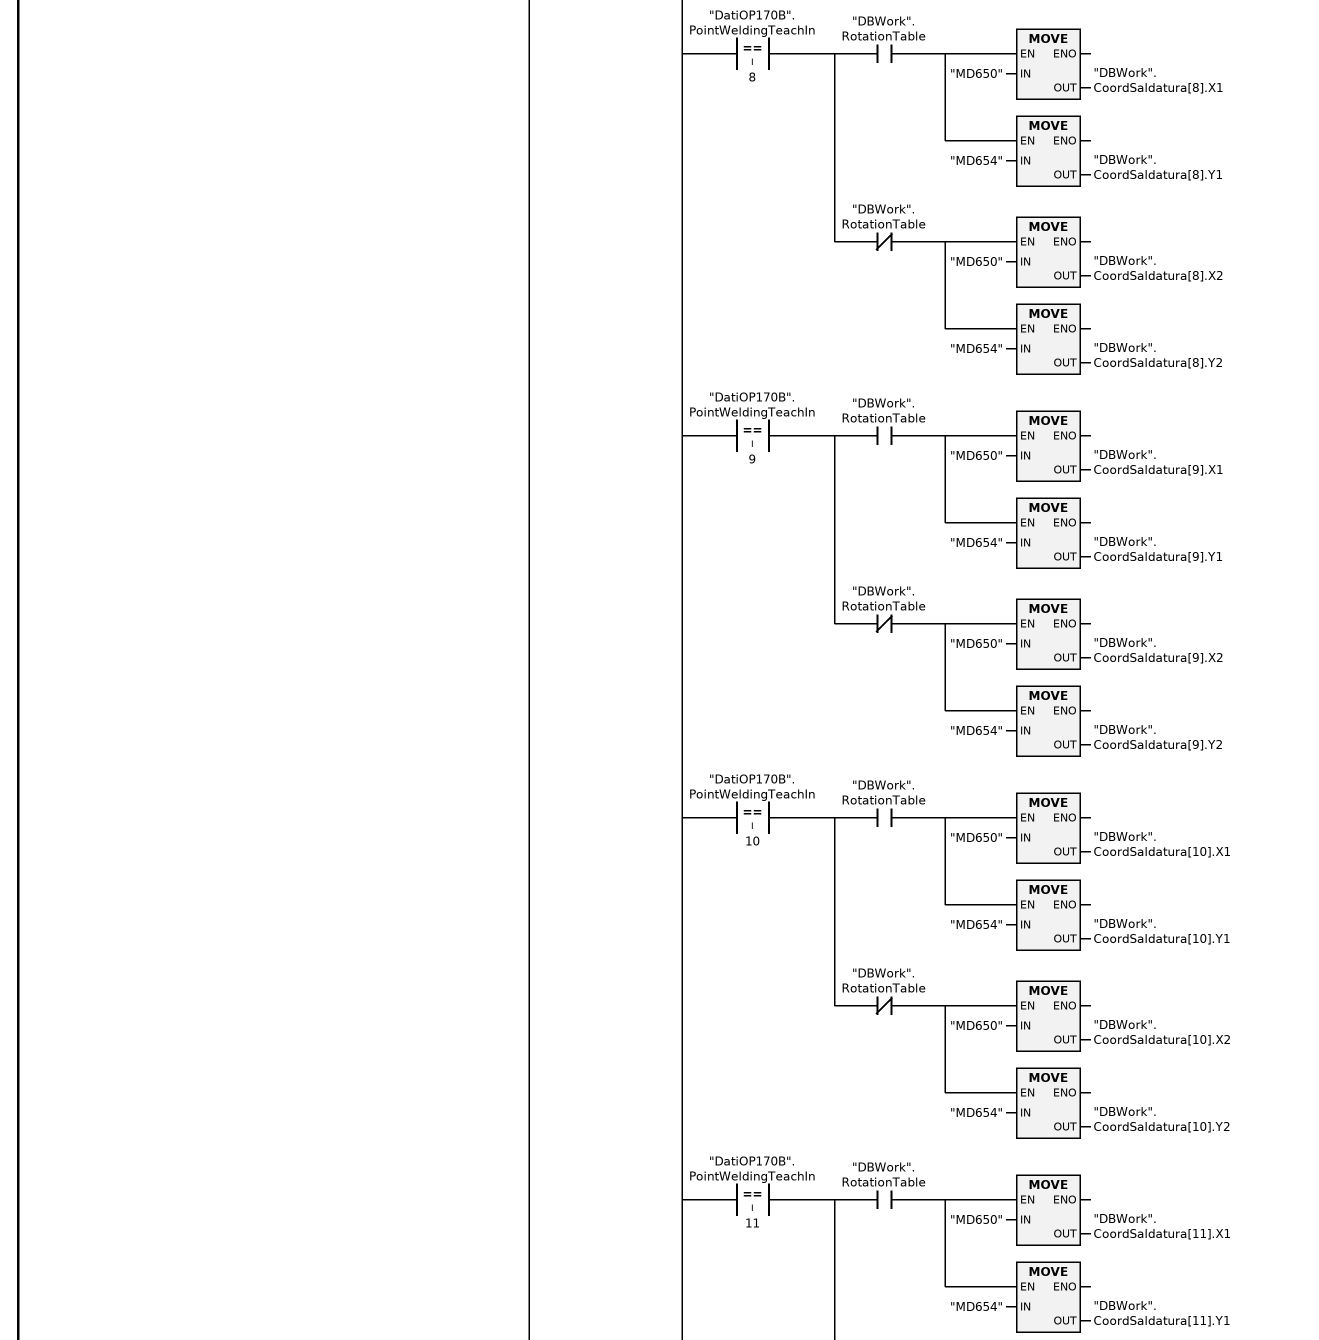
[picture p145: FC50 - TEACH-IN networks 7-7]
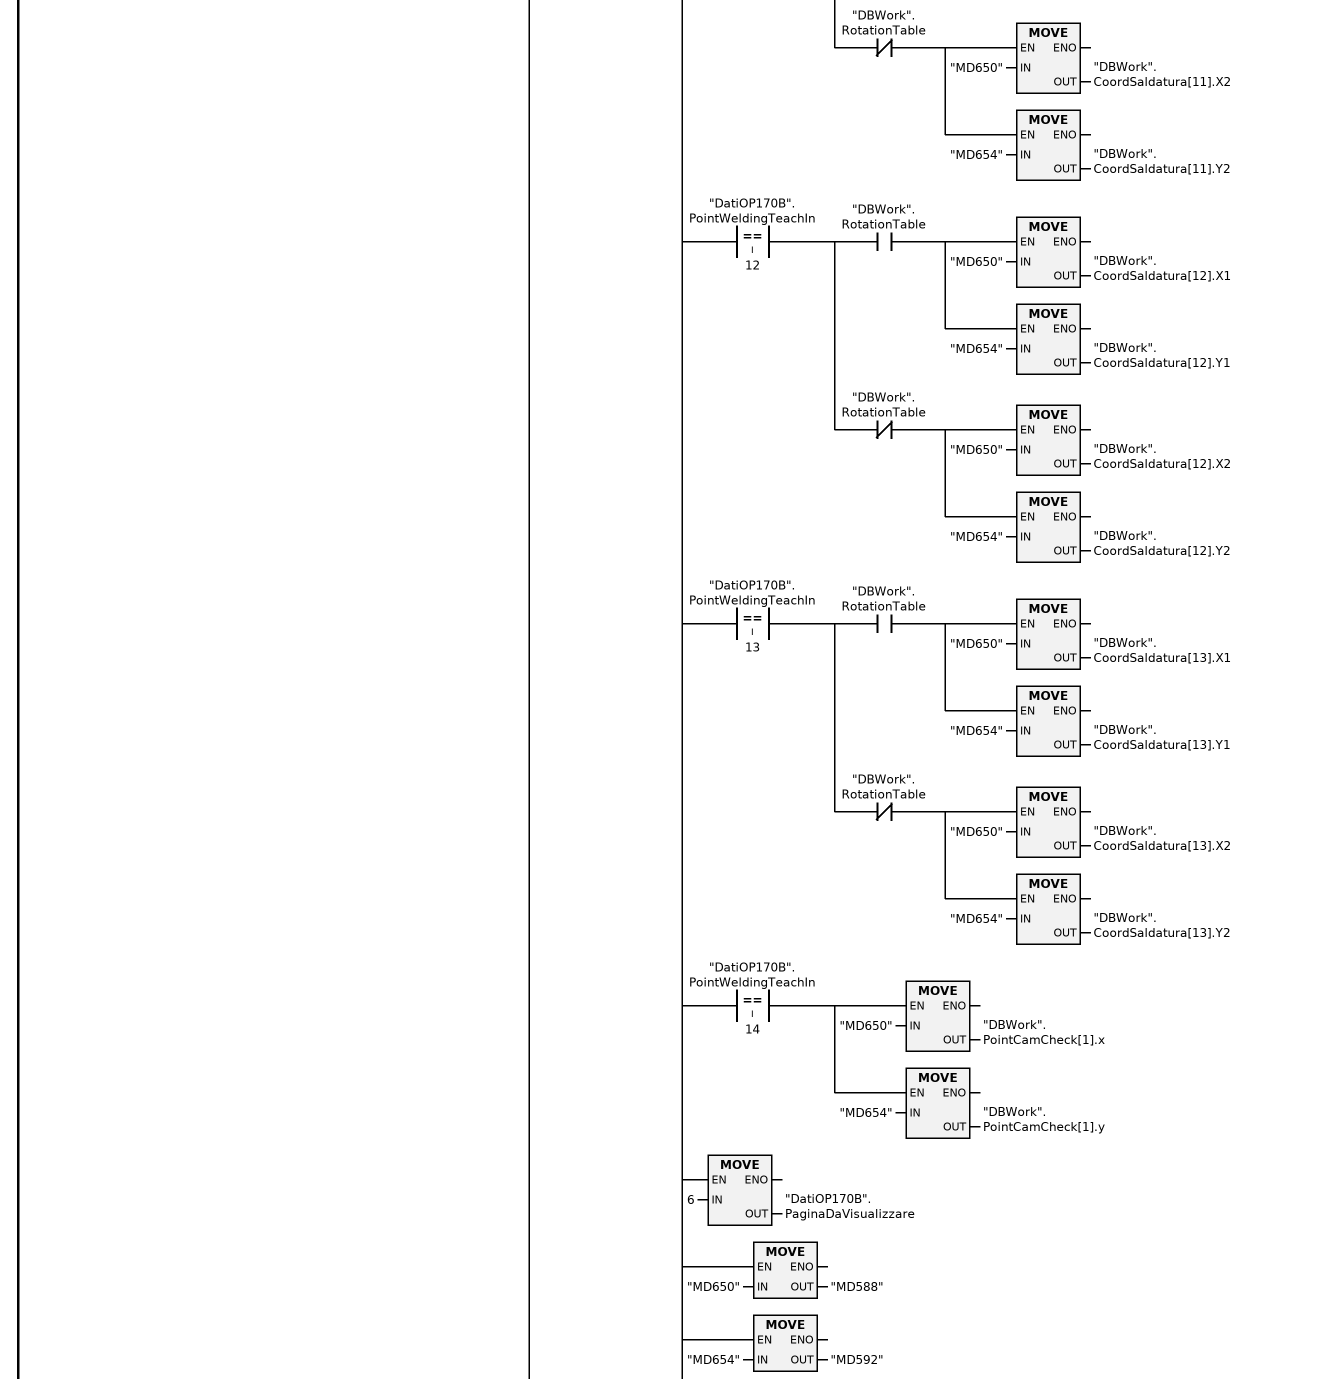
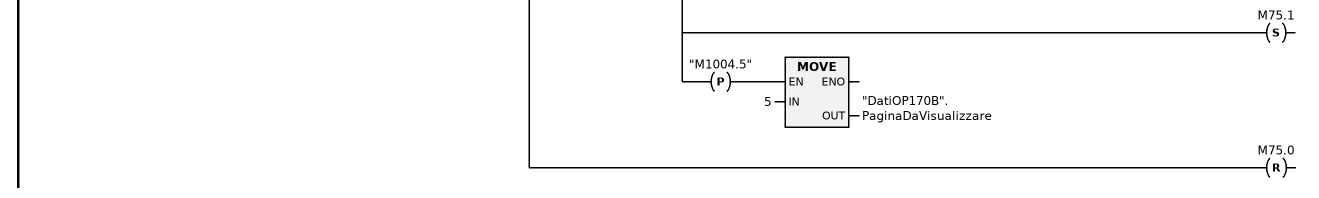
NETWORK
TITLE = Enable movement for axis on Teach-in
//move on welding point or wiev point and stored date when press teach in
//
      A     "M11.2";
      A(;
      O(;
      L     "DatiOP170B".NumeroPagina.NumeroPaginaCorrente;
      L     6;
      ==I;
      );
      O     "T63";
      );
      AN    "M346.1";
      AN    "M340.1";
      A     "M347.3";
      A     "M341.3";
      =     L 0.0;
      A     L 0.0;
      A     "T63";
      FP    "M1004.4";
      =     L 0.1;
      A     L 0.1;
      A(;
      L     "DatiOP170B".PointWeldingTeachIn;
      L     1;
      ==I;
      );
      =     L 0.2;
      A     L 0.2;
      A     "DBWork".RotationTable;
      =     L 0.3;
      A     L 0.3;
      JNB   _008;
      L     "MD650";
      T     "DBWork".CoordSaldatura[1].X1;
_008: NOP   0;
      A     L 0.3;
      JNB   _009;
      L     "MD654";
      T     "DBWork".CoordSaldatura[1].Y1;
_009: NOP   0;
      A     L 0.2;
      AN    "DBWork".RotationTable;
      =     L 0.3;
      A     L 0.3;
      JNB   _00a;
      L     "MD650";
      T     "DBWork".CoordSaldatura[1].X2;
_00a: NOP   0;
      A     L 0.3;
      JNB   _00b;
      L     "MD654";
      T     "DBWork".CoordSaldatura[1].Y2;
_00b: NOP   0;
      A     L 0.1;
      A(;
      L     "DatiOP170B".PointWeldingTeachIn;
      L     2;
      ==I;
      );
      =     L 0.2;
      A     L 0.2;
      A     "DBWork".RotationTable;
      =     L 0.3;
      A     L 0.3;
      JNB   _00c;
      L     "MD650";
      T     "DBWork".CoordSaldatura[2].X1;
_00c: NOP   0;
      A     L 0.3;
      JNB   _00d;
      L     "MD654";
      T     "DBWork".CoordSaldatura[2].Y1;
_00d: NOP   0;
      A     L 0.2;
      AN    "DBWork".RotationTable;
      =     L 0.3;
      A     L 0.3;
      JNB   _00e;
      L     "MD650";
      T     "DBWork".CoordSaldatura[2].X2;
_00e: NOP   0;
      A     L 0.3;
      JNB   _00f;
      L     "MD654";
      T     "DBWork".CoordSaldatura[2].Y2;
_00f: NOP   0;
      A     L 0.1;
      A(;
      L     "DatiOP170B".PointWeldingTeachIn;
      L     3;
      ==I;
      );
      =     L 0.2;
      A     L 0.2;
      A     "DBWork".RotationTable;
      =     L 0.3;
      A     L 0.3;
      JNB   _010;
      L     "MD650";
      T     "DBWork".CoordSaldatura[3].X1;
_010: NOP   0;
      A     L 0.3;
      JNB   _011;
      L     "MD654";
      T     "DBWork".CoordSaldatura[3].Y1;
_011: NOP   0;
      A     L 0.2;
      AN    "DBWork".RotationTable;
      =     L 0.3;
      A     L 0.3;
      JNB   _012;
      L     "MD650";
      T     "DBWork".CoordSaldatura[3].X2;
_012: NOP   0;
      A     L 0.3;
      JNB   _013;
      L     "MD654";
      T     "DBWork".CoordSaldatura[3].Y2;
_013: NOP   0;
      A     L 0.1;
      A(;
      L     "DatiOP170B".PointWeldingTeachIn;
      L     4;
      ==I;
      );
      =     L 0.2;
      A     L 0.2;
      A     "DBWork".RotationTable;
      =     L 0.3;
      A     L 0.3;
      JNB   _014;
      L     "MD650";
      T     "DBWork".CoordSaldatura[4].X1;
_014: NOP   0;
      A     L 0.3;
      JNB   _015;
      L     "MD654";
      T     "DBWork".CoordSaldatura[4].Y1;
_015: NOP   0;
      A     L 0.2;
      AN    "DBWork".RotationTable;
      =     L 0.3;
      A     L 0.3;
      JNB   _016;
      L     "MD650";
      T     "DBWork".CoordSaldatura[4].X2;
_016: NOP   0;
      A     L 0.3;
      JNB   _017;
      L     "MD654";
      T     "DBWork".CoordSaldatura[4].Y2;
_017: NOP   0;
      A     L 0.1;
      A(;
      L     "DatiOP170B".PointWeldingTeachIn;
      L     5;
      ==I;
      );
      =     L 0.2;
      A     L 0.2;
      A     "DBWork".RotationTable;
      =     L 0.3;
      A     L 0.3;
      JNB   _018;
      L     "MD650";
      T     "DBWork".CoordSaldatura[5].X1;
_018: NOP   0;
      A     L 0.3;
      JNB   _019;
      L     "MD654";
      T     "DBWork".CoordSaldatura[5].Y1;
_019: NOP   0;
      A     L 0.2;
      AN    "DBWork".RotationTable;
      =     L 0.3;
      A     L 0.3;
      JNB   _01a;
      L     "MD650";
      T     "DBWork".CoordSaldatura[5].X2;
_01a: NOP   0;
      A     L 0.3;
      JNB   _01b;
      L     "MD654";
      T     "DBWork".CoordSaldatura[5].Y2;
_01b: NOP   0;
      A     L 0.1;
      A(;
      L     "DatiOP170B".PointWeldingTeachIn;
      L     6;
      ==I;
      );
      =     L 0.2;
      A     L 0.2;
      A     "DBWork".RotationTable;
      =     L 0.3;
      A     L 0.3;
      JNB   _01c;
      L     "MD650";
      T     "DBWork".CoordSaldatura[6].X1;
_01c: NOP   0;
      A     L 0.3;
      JNB   _01d;
      L     "MD654";
      T     "DBWork".CoordSaldatura[6].Y1;
_01d: NOP   0;
      A     L 0.2;
      AN    "DBWork".RotationTable;
      =     L 0.3;
      A     L 0.3;
      JNB   _01e;
      L     "MD650";
      T     "DBWork".CoordSaldatura[6].X2;
_01e: NOP   0;
      A     L 0.3;
      JNB   _01f;
      L     "MD654";
      T     "DBWork".CoordSaldatura[6].Y2;
_01f: NOP   0;
      A     L 0.1;
      A(;
      L     "DatiOP170B".PointWeldingTeachIn;
      L     7;
      ==I;
      );
      =     L 0.2;
      A     L 0.2;
      A     "DBWork".RotationTable;
      =     L 0.3;
      A     L 0.3;
      JNB   _020;
      L     "MD650";
      T     "DBWork".CoordSaldatura[7].X1;
_020: NOP   0;
      A     L 0.3;
      JNB   _021;
      L     "MD654";
      T     "DBWork".CoordSaldatura[7].Y1;
_021: NOP   0;
      A     L 0.2;
      AN    "DBWork".RotationTable;
      =     L 0.3;
      A     L 0.3;
      JNB   _022;
      L     "MD650";
      T     "DBWork".CoordSaldatura[7].X2;
_022: NOP   0;
      A     L 0.3;
      JNB   _023;
      L     "MD654";
      T     "DBWork".CoordSaldatura[7].Y2;
_023: NOP   0;
      A     L 0.1;
      A(;
      L     "DatiOP170B".PointWeldingTeachIn;
      L     8;
      ==I;
      );
      =     L 0.2;
      A     L 0.2;
      A     "DBWork".RotationTable;
      =     L 0.3;
      A     L 0.3;
      JNB   _024;
      L     "MD650";
      T     "DBWork".CoordSaldatura[8].X1;
_024: NOP   0;
      A     L 0.3;
      JNB   _025;
      L     "MD654";
      T     "DBWork".CoordSaldatura[8].Y1;
_025: NOP   0;
      A     L 0.2;
      AN    "DBWork".RotationTable;
      =     L 0.3;
      A     L 0.3;
      JNB   _026;
      L     "MD650";
      T     "DBWork".CoordSaldatura[8].X2;
_026: NOP   0;
      A     L 0.3;
      JNB   _027;
      L     "MD654";
      T     "DBWork".CoordSaldatura[8].Y2;
_027: NOP   0;
      A     L 0.1;
      A(;
      L     "DatiOP170B".PointWeldingTeachIn;
      L     9;
      ==I;
      );
      =     L 0.2;
      A     L 0.2;
      A     "DBWork".RotationTable;
      =     L 0.3;
      A     L 0.3;
      JNB   _028;
      L     "MD650";
      T     "DBWork".CoordSaldatura[9].X1;
_028: NOP   0;
      A     L 0.3;
      JNB   _029;
      L     "MD654";
      T     "DBWork".CoordSaldatura[9].Y1;
_029: NOP   0;
      A     L 0.2;
      AN    "DBWork".RotationTable;
      =     L 0.3;
      A     L 0.3;
      JNB   _02a;
      L     "MD650";
      T     "DBWork".CoordSaldatura[9].X2;
_02a: NOP   0;
      A     L 0.3;
      JNB   _02b;
      L     "MD654";
      T     "DBWork".CoordSaldatura[9].Y2;
_02b: NOP   0;
      A     L 0.1;
      A(;
      L     "DatiOP170B".PointWeldingTeachIn;
      L     10;
      ==I;
      );
      =     L 0.2;
      A     L 0.2;
      A     "DBWork".RotationTable;
      =     L 0.3;
      A     L 0.3;
      JNB   _02c;
      L     "MD650";
      T     "DBWork".CoordSaldatura[10].X1;
_02c: NOP   0;
      A     L 0.3;
      JNB   _02d;
      L     "MD654";
      T     "DBWork".CoordSaldatura[10].Y1;
_02d: NOP   0;
      A     L 0.2;
      AN    "DBWork".RotationTable;
      =     L 0.3;
      A     L 0.3;
      JNB   _02e;
      L     "MD650";
      T     "DBWork".CoordSaldatura[10].X2;
_02e: NOP   0;
      A     L 0.3;
      JNB   _02f;
      L     "MD654";
      T     "DBWork".CoordSaldatura[10].Y2;
_02f: NOP   0;
      A     L 0.1;
      A(;
      L     "DatiOP170B".PointWeldingTeachIn;
      L     11;
      ==I;
      );
      =     L 0.2;
      A     L 0.2;
      A     "DBWork".RotationTable;
      =     L 0.3;
      A     L 0.3;
      JNB   _030;
      L     "MD650";
      T     "DBWork".CoordSaldatura[11].X1;
_030: NOP   0;
      A     L 0.3;
      JNB   _031;
      L     "MD654";
      T     "DBWork".CoordSaldatura[11].Y1;
_031: NOP   0;
      A     L 0.2;
      AN    "DBWork".RotationTable;
      =     L 0.3;
      A     L 0.3;
      JNB   _032;
      L     "MD650";
      T     "DBWork".CoordSaldatura[11].X2;
_032: NOP   0;
      A     L 0.3;
      JNB   _033;
      L     "MD654";
      T     "DBWork".CoordSaldatura[11].Y2;
_033: NOP   0;
      A     L 0.1;
      A(;
      L     "DatiOP170B".PointWeldingTeachIn;
      L     12;
      ==I;
      );
      =     L 0.2;
      A     L 0.2;
      A     "DBWork".RotationTable;
      =     L 0.3;
      A     L 0.3;
      JNB   _034;
      L     "MD650";
      T     "DBWork".CoordSaldatura[12].X1;
_034: NOP   0;
      A     L 0.3;
      JNB   _035;
      L     "MD654";
      T     "DBWork".CoordSaldatura[12].Y1;
_035: NOP   0;
      A     L 0.2;
      AN    "DBWork".RotationTable;
      =     L 0.3;
      A     L 0.3;
      JNB   _036;
      L     "MD650";
      T     "DBWork".CoordSaldatura[12].X2;
_036: NOP   0;
      A     L 0.3;
      JNB   _037;
      L     "MD654";
      T     "DBWork".CoordSaldatura[12].Y2;
_037: NOP   0;
      A     L 0.1;
      A(;
      L     "DatiOP170B".PointWeldingTeachIn;
      L     13;
      ==I;
      );
      =     L 0.2;
      A     L 0.2;
      A     "DBWork".RotationTable;
      =     L 0.3;
      A     L 0.3;
      JNB   _038;
      L     "MD650";
      T     "DBWork".CoordSaldatura[13].X1;
_038: NOP   0;
      A     L 0.3;
      JNB   _039;
      L     "MD654";
      T     "DBWork".CoordSaldatura[13].Y1;
_039: NOP   0;
      A     L 0.2;
      AN    "DBWork".RotationTable;
      =     L 0.3;
      A     L 0.3;
      JNB   _03a;
      L     "MD650";
      T     "DBWork".CoordSaldatura[13].X2;
_03a: NOP   0;
      A     L 0.3;
      JNB   _03b;
      L     "MD654";
      T     "DBWork".CoordSaldatura[13].Y2;
_03b: NOP   0;
      A     L 0.1;
      A(;
      L     "DatiOP170B".PointWeldingTeachIn;
      L     14;
      ==I;
      );
      =     L 0.2;
      A     L 0.2;
      JNB   _03c;
      L     "MD650";
      T     "DBWork".PointCamCheck[1].x;
_03c: NOP   0;
      A     L 0.2;
      JNB   _03d;
      L     "MD654";
      T     "DBWork".PointCamCheck[1].y;
_03d: NOP   0;
      A     L 0.1;
      JNB   _03e;
      L     6;
      T     "DatiOP170B".PaginaDaVisualizzare;
_03e: NOP   0;
      A     L 0.1;
      JNB   _03f;
      L     "MD650";
      T     "MD588";
_03f: NOP   0;
      A     L 0.1;
      JNB   _040;
      L     "MD654";
      T     "MD592";
_040: NOP   0;
      A     L 0.1;
      BLD   102;
      S     "M75.1";
      A     L 0.1;
      FP    "M1004.5";
      JNB   _041;
      L     5;
      T     "DatiOP170B".PaginaDaVisualizzare;
_041: NOP   0;
      A     L 0.0;
      BLD   102;
      R     "M75.0";
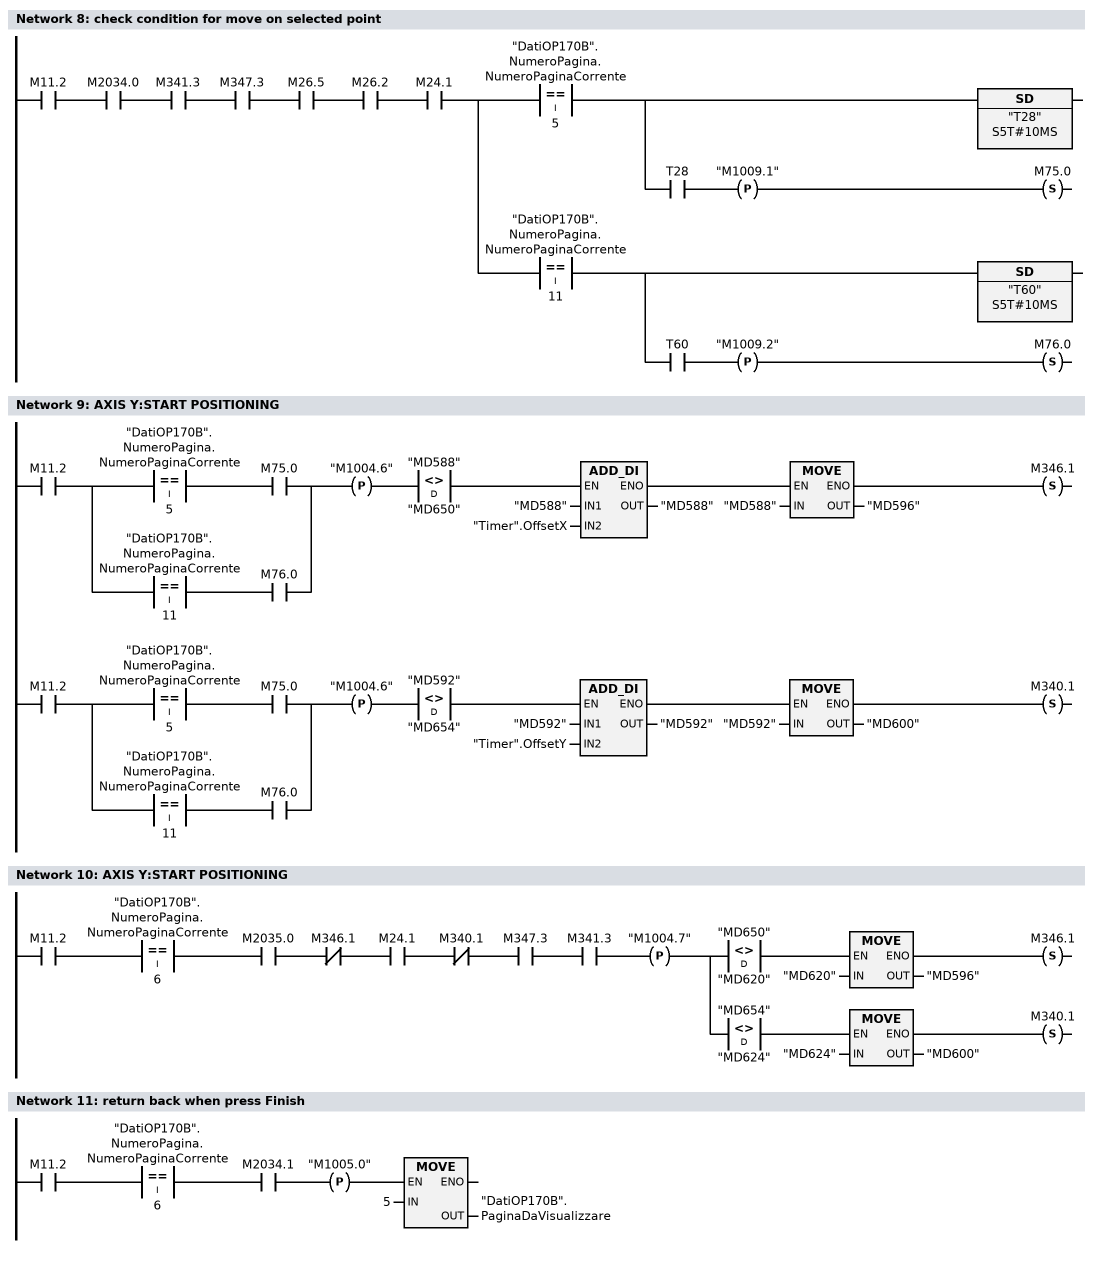
NETWORK
TITLE = check condition for move on selected point
//condition for move on selected point
      A     "M11.2";
      A     "M2034.0";
      A     "M341.3";
      A     "M347.3";
      A     "M26.5";
      A     "M26.2";
      A     "M24.1";
      =     L 1.0;
      A     L 1.0;
      A(;
      L     "DatiOP170B".NumeroPagina.NumeroPaginaCorrente;
      L     5;
      ==I;
      );
      =     L 1.1;
      A     L 1.1;
      BLD   102;
      L     S5T#10MS;
      SD    "T28";
      A     L 1.1;
      A     "T28";
      FP    "M1009.1";
      S     "M75.0";
      A     L 1.0;
      A(;
      L     "DatiOP170B".NumeroPagina.NumeroPaginaCorrente;
      L     11;
      ==I;
      );
      =     L 1.1;
      A     L 1.1;
      BLD   102;
      L     S5T#10MS;
      SD    "T60";
      A     L 1.1;
      A     "T60";
      FP    "M1009.2";
      S     "M76.0";
NETWORK
TITLE = AXIS Y:START POSITIONING
//move axis on selected point
      A     "M11.2";
      A(;
      A(;
      L     "DatiOP170B".NumeroPagina.NumeroPaginaCorrente;
      L     5;
      ==I;
      );
      A     "M75.0";
      O;
      A(;
      L     "DatiOP170B".NumeroPagina.NumeroPaginaCorrente;
      L     11;
      ==I;
      );
      A     "M76.0";
      );
      FP    "M1004.6";
      =     L 1.0;
      A(;
      A     L 1.0;
      A(;
      L     "MD588";
      L     "MD650";
      <>D;
      );
      JNB   _042;
      L     "MD588";
      L     "Timer".OffsetX;
      +D;
      T     "MD588";
      AN    OV;
      SAVE;
      CLR;
_042: A     BR;
      );
      JNB   _043;
      L     "MD588";
      T     "MD596";
      SET;
      SAVE;
      CLR;
_043: A     BR;
      S     "M346.1";
      A(;
      A     L 1.0;
      A(;
      L     "MD592";
      L     "MD654";
      <>D;
      );
      JNB   _044;
      L     "MD592";
      L     "Timer".OffsetY;
      +D;
      T     "MD592";
      AN    OV;
      SAVE;
      CLR;
_044: A     BR;
      );
      JNB   _045;
      L     "MD592";
      T     "MD600";
      SET;
      SAVE;
      CLR;
_045: A     BR;
      S     "M340.1";
NETWORK
TITLE = AXIS Y:START POSITIONING
      A     "M11.2";
      A(;
      L     "DatiOP170B".NumeroPagina.NumeroPaginaCorrente;
      L     6;
      ==I;
      );
      A     "M2035.0";
      AN    "M346.1";
      A     "M24.1";
      AN    "M340.1";
      A     "M347.3";
      A     "M341.3";
      FP    "M1004.7";
      =     L 0.0;
      A     L 0.0;
      A(;
      L     "MD650";
      L     "MD620";
      <>D;
      );
      JNB   _046;
      L     "MD620";
      T     "MD596";
      SET;
      SAVE;
      CLR;
_046: A     BR;
      S     "M346.1";
      A     L 0.0;
      A(;
      L     "MD654";
      L     "MD624";
      <>D;
      );
      JNB   _047;
      L     "MD624";
      T     "MD600";
      SET;
      SAVE;
      CLR;
_047: A     BR;
      S     "M340.1";
NETWORK
TITLE = return back when press Finish
//retirn on previus page with finish
      A     "M11.2";
      A(;
      L     "DatiOP170B".NumeroPagina.NumeroPaginaCorrente;
      L     6;
      ==I;
      );
      A     "M2034.1";
      FP    "M1005.0";
      JNB   _048;
      L     5;
      T     "DatiOP170B".PaginaDaVisualizzare;
_048: NOP   0;
END_FUNCTION

FUNCTION "FC51 - TYPE TOOL" : VOID	// FC 51
VERSION : 0.1
BEGIN
NETWORK
TITLE = 1=start read job
      A     "ChangeFunc";
      AN    "Timer".Check1;
      =     L 1.0;
      A     L 1.0;
      BLD   102;
      S     DB5.DBX 14.0;
      A     L 1.0;
      A     "Off";
      S     DB5.DBX 20.0;
NETWORK
TITLE =
NETWORK
TITLE = check if PP1 is present
//Controllo se è presente il PP1
      A(;
      AN    DB5.DBX 14.0;
      A     DB5.DBX 14.1;
      A(;
      L     DB5.DBB 16;
      L     1;
      >=I;
      );
      A(;
      L     DB5.DBB 16;
      L     5;
      <=I;
      );
      O     "Timer".Check1;
      );
      A(;
      L     "Timer".NumberVane;
      L     1;
      >=I;
      );
      A(;
      L     "Timer".NumberVane;
      L     5;
      <=I;
      );
      A(;
      A     "M15.6";
      A     "M15.7";
      O     "Timer".CheckComponent;
      );
      =     L 0.0;
      A     L 0.0;
      BLD   102;
      =     "Type_PP1";
      A     L 0.0;
      JNB   _001;
      L     10;
      T     "DBWork".NumeroSaldature;
_001: NOP   0;
NETWORK
TITLE = check if PP2 is present
//Controllo se è presente il PP2
      A(;
      AN    DB5.DBX 14.0;
      A     DB5.DBX 14.1;
      A(;
      L     DB5.DBB 16;
      L     6;
      >=I;
      );
      A(;
      L     DB5.DBB 16;
      L     10;
      <=I;
      );
      O     "Timer".Check1;
      );
      A(;
      L     "Timer".NumberVane;
      L     6;
      >=I;
      );
      A(;
      L     "Timer".NumberVane;
      L     10;
      <=I;
      );
      A(;
      A     "M15.6";
      AN    "M15.7";
      O     "Timer".CheckComponent;
      O     "On";
      );
      =     L 0.0;
      A     L 0.0;
      BLD   102;
      =     "Type_PP2";
      A     L 0.0;
      JNB   _002;
      L     11;
      T     "DBWork".NumeroSaldature;
_002: NOP   0;
NETWORK
TITLE = check if PP3 is present
//Controllo se è presente il PP3
      A(;
      AN    DB5.DBX 14.0;
      A     DB5.DBX 14.1;
      A(;
      L     DB5.DBB 16;
      L     11;
      >=I;
      );
      A(;
      L     DB5.DBB 16;
      L     15;
      <=I;
      );
      O     "Timer".Check1;
      );
      A(;
      L     "Timer".NumberVane;
      L     11;
      >=I;
      );
      A(;
      L     "Timer".NumberVane;
      L     15;
      <=I;
      );
      A(;
      AN    "M15.6";
      A     "M15.7";
      O     "Timer".CheckComponent;
      );
      =     L 0.0;
      A     L 0.0;
      BLD   102;
      =     "Type_PP3";
      A     L 0.0;
      JNB   _003;
      L     9;
      T     "DBWork".NumeroSaldature;
_003: NOP   0;
NETWORK
TITLE = check if PP4 is present
//Controllo se è presente il PP4
      A(;
      AN    DB5.DBX 14.0;
      A     DB5.DBX 14.1;
      A(;
      L     DB5.DBB 16;
      L     16;
      >=I;
      );
      A(;
      L     DB5.DBB 16;
      L     20;
      <=I;
      );
      O     "Timer".Check1;
      );
      A(;
      L     "Timer".NumberVane;
      L     16;
      >=I;
      );
      A(;
      L     "Timer".NumberVane;
      L     20;
      <=I;
      );
      A(;
      AN    "M15.6";
      AN    "M15.7";
      O     "Timer".CheckComponent;
      );
      =     L 0.0;
      A     L 0.0;
      BLD   102;
      =     "Type_PP4";
      A     L 0.0;
      JNB   _004;
      L     13;
      T     "DBWork".NumeroSaldature;
_004: NOP   0;
NETWORK
TITLE = timer for change value
      A     "ChangeFunc";
      L     S5T#1S;
      SE    "T45";
NETWORK
TITLE = load on DBWork value for weldind point PP1
//Carico sul DB Work le cordinate dei punti da saldare per il PP1
      A     "Type_PP1";
      A     "T45";
      =     L 1.0;
      A     L 1.0;
      A     "On";
      A(;
      L     "Timer".NumberVane;
      L     1;
      ==I;
      );
      =     L 1.1;
      A     L 1.1;
      JNB   _005;
      CALL  "BLKMOV" (
           SRCBLK                   := "coordinate".CoordSaldaturaPP1,
           RET_VAL                  := MW 2044,
           DSTBLK                   := "DBWork".CoordSaldatura);
_005: NOP   0;
      A     L 1.1;
      JNB   _006;
      L     "coordinate".NumeroSaldaturePP1;
      T     "DBWork".NumeroSaldature;
_006: NOP   0;
      A     L 1.1;
      JNB   _007;
      L     "coordinate".CoordinateCam_PP1[1].X;
      T     "DBWork".PointCamCheck[1].x;
_007: NOP   0;
      A     L 1.1;
      JNB   _008;
      L     "coordinate".CoordinateCam_PP1[1].Y;
      T     "DBWork".PointCamCheck[1].y;
_008: NOP   0;
      A     L 1.1;
      JNB   _009;
      L     "coordinate".CoordinateCam_PP1[2].X;
      T     "DBWork".PointCamCheck[2].x;
_009: NOP   0;
      A     L 1.1;
      JNB   _00a;
      L     "coordinate".CoordinateCam_PP1[2].Y;
      T     "DBWork".PointCamCheck[2].y;
_00a: NOP   0;
      A     L 1.1;
      JNB   _00b;
      L     "coordinate".TimeWeldingPP1[1];
      T     "DBWork".TempoSaldatura[1];
_00b: NOP   0;
      A     L 1.1;
      JNB   _00c;
      L     "coordinate".TimeWeldingPP1[2];
      T     "DBWork".TempoSaldatura[2];
_00c: NOP   0;
      A     L 1.0;
      A     "On";
      A(;
      L     "Timer".NumberVane;
      L     2;
      ==I;
      );
      =     L 1.1;
      A     L 1.1;
      JNB   _00d;
      CALL  "BLKMOV" (
           SRCBLK                   := "coordinate".CoordSaldaturaPP2,
           RET_VAL                  := MW 2044,
           DSTBLK                   := "DBWork".CoordSaldatura);
_00d: NOP   0;
      A     L 1.1;
      JNB   _00e;
      L     "coordinate".NumeroSaldaturePP2;
      T     "DBWork".NumeroSaldature;
_00e: NOP   0;
      A     L 1.1;
      JNB   _00f;
      L     "coordinate".CoordinateCam_PP2[1].X;
      T     "DBWork".PointCamCheck[1].x;
_00f: NOP   0;
      A     L 1.1;
      JNB   _010;
      L     "coordinate".CoordinateCam_PP2[1].Y;
      T     "DBWork".PointCamCheck[1].y;
_010: NOP   0;
      A     L 1.1;
      JNB   _011;
      L     "coordinate".CoordinateCam_PP2[2].X;
      T     "DBWork".PointCamCheck[2].x;
_011: NOP   0;
      A     L 1.1;
      JNB   _012;
      L     "coordinate".CoordinateCam_PP2[2].Y;
      T     "DBWork".PointCamCheck[2].y;
_012: NOP   0;
      A     L 1.1;
      JNB   _013;
      L     "coordinate".TimeWeldingPP2[1];
      T     "DBWork".TempoSaldatura[1];
_013: NOP   0;
      A     L 1.1;
      JNB   _014;
      L     "coordinate".TimeWeldingPP2[2];
      T     "DBWork".TempoSaldatura[2];
_014: NOP   0;
      A     L 1.0;
      A     "On";
      A(;
      L     "Timer".NumberVane;
      L     3;
      ==I;
      );
      =     L 1.1;
      A     L 1.1;
      JNB   _015;
      CALL  "BLKMOV" (
           SRCBLK                   := "coordinate".CoordSaldaturaPP3,
           RET_VAL                  := MW 2044,
           DSTBLK                   := "DBWork".CoordSaldatura);
_015: NOP   0;
      A     L 1.1;
      JNB   _016;
      L     "coordinate".NumeroSaldaturePP3;
      T     "DBWork".NumeroSaldature;
_016: NOP   0;
      A     L 1.1;
      JNB   _017;
      L     "coordinate".CoordinateCam_PP3[1].X;
      T     "DBWork".PointCamCheck[1].x;
_017: NOP   0;
      A     L 1.1;
      JNB   _018;
      L     "coordinate".CoordinateCam_PP3[1].Y;
      T     "DBWork".PointCamCheck[1].y;
_018: NOP   0;
      A     L 1.1;
      JNB   _019;
      L     "coordinate".CoordinateCam_PP3[2].X;
      T     "DBWork".PointCamCheck[2].x;
_019: NOP   0;
      A     L 1.1;
      JNB   _01a;
      L     "coordinate".CoordinateCam_PP3[2].Y;
      T     "DBWork".PointCamCheck[2].y;
_01a: NOP   0;
      A     L 1.1;
      JNB   _01b;
      L     "coordinate".TimeWeldingPP3[1];
      T     "DBWork".TempoSaldatura[1];
_01b: NOP   0;
      A     L 1.1;
      JNB   _01c;
      L     "coordinate".TimeWeldingPP3[2];
      T     "DBWork".TempoSaldatura[2];
_01c: NOP   0;
      A     L 1.0;
      A     "On";
      A(;
      L     "Timer".NumberVane;
      L     4;
      ==I;
      );
      =     L 1.1;
      A     L 1.1;
      JNB   _01d;
      CALL  "BLKMOV" (
           SRCBLK                   := "coordinate".CoordSaldaturaPP4,
           RET_VAL                  := MW 2044,
           DSTBLK                   := "DBWork".CoordSaldatura);
_01d: NOP   0;
      A     L 1.1;
      JNB   _01e;
      L     "coordinate".NumeroSaldaturePP4;
      T     "DBWork".NumeroSaldature;
_01e: NOP   0;
      A     L 1.1;
      JNB   _01f;
      L     "coordinate".CoordinateCam_PP4[1].X;
      T     "DBWork".PointCamCheck[1].x;
_01f: NOP   0;
      A     L 1.1;
      JNB   _020;
      L     "coordinate".CoordinateCam_PP4[1].Y;
      T     "DBWork".PointCamCheck[1].y;
_020: NOP   0;
      A     L 1.1;
      JNB   _021;
      L     "coordinate".CoordinateCam_PP4[2].X;
      T     "DBWork".PointCamCheck[2].x;
_021: NOP   0;
      A     L 1.1;
      JNB   _022;
      L     "coordinate".CoordinateCam_PP4[2].Y;
      T     "DBWork".PointCamCheck[2].y;
_022: NOP   0;
      A     L 1.1;
      JNB   _023;
      L     "coordinate".TimeWeldingPP4[1];
      T     "DBWork".TempoSaldatura[1];
_023: NOP   0;
      A     L 1.1;
      JNB   _024;
      L     "coordinate".TimeWeldingPP4[2];
      T     "DBWork".TempoSaldatura[2];
_024: NOP   0;
      A     L 1.0;
      A     "On";
      A(;
      L     "Timer".NumberVane;
      L     5;
      ==I;
      );
      =     L 1.1;
      A     L 1.1;
      JNB   _025;
      CALL  "BLKMOV" (
           SRCBLK                   := "coordinate".CoordSaldaturaPP5,
           RET_VAL                  := MW 2044,
           DSTBLK                   := "DBWork".CoordSaldatura);
_025: NOP   0;
      A     L 1.1;
      JNB   _026;
      L     "coordinate".NumeroSaldaturePP5;
      T     "DBWork".NumeroSaldature;
_026: NOP   0;
      A     L 1.1;
      JNB   _027;
      L     "coordinate".CoordinateCam_PP5[1].X;
      T     "DBWork".PointCamCheck[1].x;
_027: NOP   0;
      A     L 1.1;
      JNB   _028;
      L     "coordinate".CoordinateCam_PP5[1].Y;
      T     "DBWork".PointCamCheck[1].y;
_028: NOP   0;
      A     L 1.1;
      JNB   _029;
      L     "coordinate".CoordinateCam_PP5[2].X;
      T     "DBWork".PointCamCheck[2].x;
_029: NOP   0;
      A     L 1.1;
      JNB   _02a;
      L     "coordinate".CoordinateCam_PP5[2].Y;
      T     "DBWork".PointCamCheck[2].y;
_02a: NOP   0;
      A     L 1.1;
      JNB   _02b;
      L     "coordinate".TimeWeldingPP5[1];
      T     "DBWork".TempoSaldatura[1];
_02b: NOP   0;
      A     L 1.1;
      JNB   _02c;
      L     "coordinate".TimeWeldingPP5[2];
      T     "DBWork".TempoSaldatura[2];
_02c: NOP   0;
NETWORK
TITLE = load on DBWork value for weldind point PP2
//Carico sul DB Work le cordinate dei punti da saldare per il PP2
      A     "Type_PP2";
      A     "T45";
      =     L 1.0;
      A     L 1.0;
      A     "On";
      A(;
      L     "Timer".NumberVane;
      L     6;
      ==I;
      );
      =     L 1.1;
      A     L 1.1;
      JNB   _02d;
      CALL  "BLKMOV" (
           SRCBLK                   := "coordinate".CoordSaldaturaPP6,
           RET_VAL                  := MW 2044,
           DSTBLK                   := "DBWork".CoordSaldatura);
_02d: NOP   0;
      A     L 1.1;
      JNB   _02e;
      L     "coordinate".NumeroSaldaturePP6;
      T     "DBWork".NumeroSaldature;
_02e: NOP   0;
      A     L 1.1;
      JNB   _02f;
      L     "coordinate".CoordinateCam_PP6[1].X;
      T     "DBWork".PointCamCheck[1].x;
_02f: NOP   0;
      A     L 1.1;
      JNB   _030;
      L     "coordinate".CoordinateCam_PP6[1].Y;
      T     "DBWork".PointCamCheck[1].y;
_030: NOP   0;
      A     L 1.1;
      JNB   _031;
      L     "coordinate".TimeWeldingPP6[1];
      T     "DBWork".TempoSaldatura[1];
_031: NOP   0;
      A     L 1.1;
      JNB   _032;
      L     "coordinate".TimeWeldingPP6[2];
      T     "DBWork".TempoSaldatura[2];
_032: NOP   0;
      A     L 1.0;
      A     "On";
      A(;
      L     "Timer".NumberVane;
      L     7;
      ==I;
      );
      =     L 1.1;
      A     L 1.1;
      JNB   _033;
      CALL  "BLKMOV" (
           SRCBLK                   := "coordinate".CoordSaldaturaPP7,
           RET_VAL                  := MW 2044,
           DSTBLK                   := "DBWork".CoordSaldatura);
_033: NOP   0;
      A     L 1.1;
      JNB   _034;
      L     "coordinate".NumeroSaldaturePP7;
      T     "DBWork".NumeroSaldature;
_034: NOP   0;
      A     L 1.1;
      JNB   _035;
      L     "coordinate".CoordinateCam_PP7[1].X;
      T     "DBWork".PointCamCheck[1].x;
_035: NOP   0;
      A     L 1.1;
      JNB   _036;
      L     "coordinate".CoordinateCam_PP7[1].Y;
      T     "DBWork".PointCamCheck[1].y;
_036: NOP   0;
      A     L 1.1;
      JNB   _037;
      L     "coordinate".TimeWeldingPP7[1];
      T     "DBWork".TempoSaldatura[1];
_037: NOP   0;
      A     L 1.1;
      JNB   _038;
      L     "coordinate".TimeWeldingPP7[2];
      T     "DBWork".TempoSaldatura[2];
_038: NOP   0;
      A     L 1.0;
      A     "On";
      A(;
      L     "Timer".NumberVane;
      L     8;
      ==I;
      );
      =     L 1.1;
      A     L 1.1;
      JNB   _039;
      CALL  "BLKMOV" (
           SRCBLK                   := "coordinate".CoordSaldaturaPP8,
           RET_VAL                  := MW 2044,
           DSTBLK                   := "DBWork".CoordSaldatura);
_039: NOP   0;
      A     L 1.1;
      JNB   _03a;
      L     "coordinate".NumeroSaldaturePP8;
      T     "DBWork".NumeroSaldature;
_03a: NOP   0;
      A     L 1.1;
      JNB   _03b;
      L     "coordinate".CoordinateCam_PP8[1].X;
      T     "DBWork".PointCamCheck[1].x;
_03b: NOP   0;
      A     L 1.1;
      JNB   _03c;
      L     "coordinate".CoordinateCam_PP8[1].Y;
      T     "DBWork".PointCamCheck[1].y;
_03c: NOP   0;
      A     L 1.1;
      JNB   _03d;
      L     "coordinate".TimeWeldingPP8[1];
      T     "DBWork".TempoSaldatura[1];
_03d: NOP   0;
      A     L 1.1;
      JNB   _03e;
      L     "coordinate".TimeWeldingPP8[2];
      T     "DBWork".TempoSaldatura[2];
_03e: NOP   0;
      A     L 1.0;
      A     "On";
      A(;
      L     "Timer".NumberVane;
      L     9;
      ==I;
      );
      =     L 1.1;
      A     L 1.1;
      JNB   _03f;
      CALL  "BLKMOV" (
           SRCBLK                   := "coordinate".CoordSaldaturaPP9,
           RET_VAL                  := MW 2044,
           DSTBLK                   := "DBWork".CoordSaldatura);
_03f: NOP   0;
      A     L 1.1;
      JNB   _040;
      L     "coordinate".NumeroSaldaturePP9;
      T     "DBWork".NumeroSaldature;
_040: NOP   0;
      A     L 1.1;
      JNB   _041;
      L     "coordinate".CoordinateCam_PP9[1].X;
      T     "DBWork".PointCamCheck[1].x;
_041: NOP   0;
      A     L 1.1;
      JNB   _042;
      L     "coordinate".CoordinateCam_PP9[1].Y;
      T     "DBWork".PointCamCheck[1].y;
_042: NOP   0;
      A     L 1.1;
      JNB   _043;
      L     "coordinate".TimeWeldingPP9[1];
      T     "DBWork".TempoSaldatura[1];
_043: NOP   0;
      A     L 1.1;
      JNB   _044;
      L     "coordinate".TimeWeldingPP9[2];
      T     "DBWork".TempoSaldatura[2];
_044: NOP   0;
      A     L 1.0;
      A     "On";
      A(;
      L     "Timer".NumberVane;
      L     10;
      ==I;
      );
      =     L 1.1;
      A     L 1.1;
      JNB   _045;
      CALL  "BLKMOV" (
           SRCBLK                   := "coordinate".CoordSaldaturaPP10,
           RET_VAL                  := MW 2044,
           DSTBLK                   := "DBWork".CoordSaldatura);
_045: NOP   0;
      A     L 1.1;
      JNB   _046;
      L     "coordinate".NumeroSaldaturePP10;
      T     "DBWork".NumeroSaldature;
_046: NOP   0;
      A     L 1.1;
      JNB   _047;
      L     "coordinate".CoordinateCam_PP10[1].X;
      T     "DBWork".PointCamCheck[1].x;
_047: NOP   0;
      A     L 1.1;
      JNB   _048;
      L     "coordinate".CoordinateCam_PP10[1].Y;
      T     "DBWork".PointCamCheck[1].y;
_048: NOP   0;
      A     L 1.1;
      JNB   _049;
      L     "coordinate".TimeWeldingPP10[1];
      T     "DBWork".TempoSaldatura[1];
_049: NOP   0;
      A     L 1.1;
      JNB   _04a;
      L     "coordinate".TimeWeldingPP10[2];
      T     "DBWork".TempoSaldatura[2];
_04a: NOP   0;
NETWORK
TITLE = load on DBWork value for weldind point PP3
//Carico sul DB Work le cordinate dei punti da saldare per il PP3
      A     "Type_PP3";
      A     "T45";
      =     L 1.0;
      A     L 1.0;
      A     "On";
      A(;
      L     "Timer".NumberVane;
      L     11;
      ==I;
      );
      =     L 1.1;
      A     L 1.1;
      JNB   _04b;
      CALL  "BLKMOV" (
           SRCBLK                   := "coordinate".CoordSaldaturaPP11,
           RET_VAL                  := MW 2044,
           DSTBLK                   := "DBWork".CoordSaldatura);
_04b: NOP   0;
      A     L 1.1;
      JNB   _04c;
      L     "coordinate".NumeroSaldaturePP11;
      T     "DBWork".NumeroSaldature;
_04c: NOP   0;
      A     L 1.1;
      JNB   _04d;
      L     "coordinate".CoordinateCam_PP11[1].X;
      T     "DBWork".PointCamCheck[1].x;
_04d: NOP   0;
      A     L 1.1;
      JNB   _04e;
      L     "coordinate".CoordinateCam_PP11[1].Y;
      T     "DBWork".PointCamCheck[1].y;
_04e: NOP   0;
      A     L 1.1;
      JNB   _04f;
      L     "coordinate".TimeWeldingPP11[1];
      T     "DBWork".TempoSaldatura[1];
_04f: NOP   0;
      A     L 1.1;
      JNB   _050;
      L     "coordinate".TimeWeldingPP11[2];
      T     "DBWork".TempoSaldatura[2];
_050: NOP   0;
      A     L 1.0;
      A     "On";
      A(;
      L     "Timer".NumberVane;
      L     12;
      ==I;
      );
      =     L 1.1;
      A     L 1.1;
      JNB   _051;
      CALL  "BLKMOV" (
           SRCBLK                   := "coordinate".CoordSaldaturaPP12,
           RET_VAL                  := MW 2044,
           DSTBLK                   := "DBWork".CoordSaldatura);
_051: NOP   0;
      A     L 1.1;
      JNB   _052;
      L     "coordinate".NumeroSaldaturePP12;
      T     "DBWork".NumeroSaldature;
_052: NOP   0;
      A     L 1.1;
      JNB   _053;
      L     "coordinate".NumeroSaldaturePP12;
      T     "DBWork".NumeroSaldature;
_053: NOP   0;
      A     L 1.1;
      JNB   _054;
      L     "coordinate".CoordinateCam_PP12[1].X;
      T     "DBWork".PointCamCheck[1].x;
_054: NOP   0;
      A     L 1.1;
      JNB   _055;
      L     "coordinate".CoordinateCam_PP12[1].Y;
      T     "DBWork".PointCamCheck[1].y;
_055: NOP   0;
      A     L 1.1;
      JNB   _056;
      L     "coordinate".TimeWeldingPP12[2];
      T     "DBWork".TempoSaldatura[2];
_056: NOP   0;
      A     L 1.0;
      A     "On";
      A(;
      L     "Timer".NumberVane;
      L     13;
      ==I;
      );
      =     L 1.1;
      A     L 1.1;
      JNB   _057;
      CALL  "BLKMOV" (
           SRCBLK                   := "coordinate".CoordSaldaturaPP13,
           RET_VAL                  := MW 2044,
           DSTBLK                   := "DBWork".CoordSaldatura);
_057: NOP   0;
      A     L 1.1;
      JNB   _058;
      L     "coordinate".NumeroSaldaturePP13;
      T     "DBWork".NumeroSaldature;
_058: NOP   0;
      A     L 1.1;
      JNB   _059;
      L     "coordinate".NumeroSaldaturePP13;
      T     "DBWork".NumeroSaldature;
_059: NOP   0;
      A     L 1.1;
      JNB   _05a;
      L     "coordinate".CoordinateCam_PP13[1].X;
      T     "DBWork".PointCamCheck[1].x;
_05a: NOP   0;
      A     L 1.1;
      JNB   _05b;
      L     "coordinate".CoordinateCam_PP13[1].Y;
      T     "DBWork".PointCamCheck[1].y;
_05b: NOP   0;
      A     L 1.1;
      JNB   _05c;
      L     "coordinate".TimeWeldingPP13[2];
      T     "DBWork".TempoSaldatura[2];
_05c: NOP   0;
      A     L 1.0;
      A     "On";
      A(;
      L     "Timer".NumberVane;
      L     14;
      ==I;
      );
      =     L 1.1;
      A     L 1.1;
      JNB   _05d;
      CALL  "BLKMOV" (
           SRCBLK                   := "coordinate".CoordSaldaturaPP14,
           RET_VAL                  := MW 2044,
           DSTBLK                   := "DBWork".CoordSaldatura);
_05d: NOP   0;
      A     L 1.1;
      JNB   _05e;
      L     "coordinate".NumeroSaldaturePP14;
      T     "DBWork".NumeroSaldature;
_05e: NOP   0;
      A     L 1.1;
      JNB   _05f;
      L     "coordinate".NumeroSaldaturePP14;
      T     "DBWork".NumeroSaldature;
_05f: NOP   0;
      A     L 1.1;
      JNB   _060;
      L     "coordinate".NumeroSaldaturePP14;
      T     "DBWork".NumeroSaldature;
_060: NOP   0;
      A     L 1.1;
      JNB   _061;
      L     "coordinate".CoordinateCam_PP14[1].X;
      T     "DBWork".PointCamCheck[1].x;
_061: NOP   0;
      A     L 1.1;
      JNB   _062;
      L     "coordinate".CoordinateCam_PP14[1].Y;
      T     "DBWork".PointCamCheck[1].y;
_062: NOP   0;
      A     L 1.1;
      JNB   _063;
      L     "coordinate".TimeWeldingPP14[2];
      T     "DBWork".TempoSaldatura[2];
_063: NOP   0;
      A     L 1.0;
      A     "On";
      A(;
      L     "Timer".NumberVane;
      L     15;
      ==I;
      );
      =     L 1.1;
      A     L 1.1;
      JNB   _064;
      CALL  "BLKMOV" (
           SRCBLK                   := "coordinate".CoordSaldaturaPP15,
           RET_VAL                  := MW 2044,
           DSTBLK                   := "DBWork".CoordSaldatura);
_064: NOP   0;
      A     L 1.1;
      JNB   _065;
      L     "coordinate".NumeroSaldaturePP15;
      T     "DBWork".NumeroSaldature;
_065: NOP   0;
      A     L 1.1;
      JNB   _066;
      L     "coordinate".NumeroSaldaturePP15;
      T     "DBWork".NumeroSaldature;
_066: NOP   0;
      A     L 1.1;
      JNB   _067;
      L     "coordinate".NumeroSaldaturePP15;
      T     "DBWork".NumeroSaldature;
_067: NOP   0;
      A     L 1.1;
      JNB   _068;
      L     "coordinate".NumeroSaldaturePP15;
      T     "DBWork".NumeroSaldature;
_068: NOP   0;
      A     L 1.1;
      JNB   _069;
      L     "coordinate".CoordinateCam_PP15[1].X;
      T     "DBWork".PointCamCheck[1].x;
_069: NOP   0;
      A     L 1.1;
      JNB   _06a;
      L     "coordinate".CoordinateCam_PP15[1].Y;
      T     "DBWork".PointCamCheck[1].y;
_06a: NOP   0;
      A     L 1.1;
      JNB   _06b;
      L     "coordinate".TimeWeldingPP15[2];
      T     "DBWork".TempoSaldatura[2];
_06b: NOP   0;
NETWORK
TITLE = load on DBWork value for weldind point PP4
//Carico sul DB Work le cordinate dei punti da saldare per il PP4
      A     "Type_PP4";
      A     "T45";
      =     L 1.0;
      A     L 1.0;
      A     "On";
      A(;
      L     "Timer".NumberVane;
      L     16;
      ==I;
      );
      =     L 1.1;
      A     L 1.1;
      JNB   _06c;
      CALL  "BLKMOV" (
           SRCBLK                   := "coordinate".CoordSaldaturaPP16,
           RET_VAL                  := MW 2044,
           DSTBLK                   := "DBWork".CoordSaldatura);
_06c: A     BR;
      S     M 465.0;
      A     L 1.1;
      JNB   _06d;
      L     "coordinate".NumeroSaldaturePP16;
      T     "DBWork".NumeroSaldature;
_06d: NOP   0;
      A     L 1.1;
      JNB   _06e;
      L     "coordinate".CoordinateCam_PP16[1].X;
      T     "DBWork".PointCamCheck[1].x;
_06e: NOP   0;
      A     L 1.1;
      JNB   _06f;
      L     "coordinate".CoordinateCam_PP16[1].Y;
      T     "DBWork".PointCamCheck[1].y;
_06f: NOP   0;
      A     L 1.1;
      JNB   _070;
      L     "coordinate".TimeWeldingPP16[1];
      T     "DBWork".TempoSaldatura[1];
_070: NOP   0;
      A     L 1.1;
      JNB   _071;
      L     "coordinate".TimeWeldingPP16[2];
      T     "DBWork".TempoSaldatura[2];
_071: NOP   0;
      A     L 1.0;
      A     "On";
      A(;
      L     "Timer".NumberVane;
      L     17;
      ==I;
      );
      =     L 1.1;
      A     L 1.1;
      JNB   _072;
      CALL  "BLKMOV" (
           SRCBLK                   := "coordinate".CoordSaldaturaPP17,
           RET_VAL                  := MW 2044,
           DSTBLK                   := "DBWork".CoordSaldatura);
_072: NOP   0;
      A     L 1.1;
      JNB   _073;
      L     "coordinate".NumeroSaldaturePP17;
      T     "DBWork".NumeroSaldature;
_073: NOP   0;
      A     L 1.1;
      JNB   _074;
      L     "coordinate".CoordinateCam_PP17[1].X;
      T     "DBWork".PointCamCheck[1].x;
_074: NOP   0;
      A     L 1.1;
      JNB   _075;
      L     "coordinate".CoordinateCam_PP17[1].Y;
      T     "DBWork".PointCamCheck[1].y;
_075: NOP   0;
      A     L 1.1;
      JNB   _076;
      L     "coordinate".TimeWeldingPP17[1];
      T     "DBWork".TempoSaldatura[1];
_076: NOP   0;
      A     L 1.1;
      JNB   _077;
      L     "coordinate".TimeWeldingPP17[2];
      T     "DBWork".TempoSaldatura[2];
_077: NOP   0;
      A     L 1.0;
      A     "On";
      A(;
      L     "Timer".NumberVane;
      L     18;
      ==I;
      );
      =     L 1.1;
      A     L 1.1;
      JNB   _078;
      CALL  "BLKMOV" (
           SRCBLK                   := "coordinate".CoordSaldaturaPP18,
           RET_VAL                  := MW 2044,
           DSTBLK                   := "DBWork".CoordSaldatura);
_078: NOP   0;
      A     L 1.1;
      JNB   _079;
      L     "coordinate".NumeroSaldaturePP18;
      T     "DBWork".NumeroSaldature;
_079: NOP   0;
      A     L 1.1;
      JNB   _07a;
      L     "coordinate".CoordinateCam_PP18[1].X;
      T     "DBWork".PointCamCheck[1].x;
_07a: NOP   0;
      A     L 1.1;
      JNB   _07b;
      L     "coordinate".CoordinateCam_PP18[1].Y;
      T     "DBWork".PointCamCheck[1].y;
_07b: NOP   0;
      A     L 1.1;
      JNB   _07c;
      L     "coordinate".TimeWeldingPP18[1];
      T     "DBWork".TempoSaldatura[1];
_07c: NOP   0;
      A     L 1.1;
      JNB   _07d;
      L     "coordinate".TimeWeldingPP18[2];
      T     "DBWork".TempoSaldatura[2];
_07d: NOP   0;
      A     L 1.0;
      A     "On";
      A(;
      L     "Timer".NumberVane;
      L     19;
      ==I;
      );
      =     L 1.1;
      A     L 1.1;
      JNB   _07e;
      CALL  "BLKMOV" (
           SRCBLK                   := "coordinate".CoordSaldaturaPP19,
           RET_VAL                  := MW 2044,
           DSTBLK                   := "DBWork".CoordSaldatura);
_07e: NOP   0;
      A     L 1.1;
      JNB   _07f;
      L     "coordinate".NumeroSaldaturePP19;
      T     "DBWork".NumeroSaldature;
_07f: NOP   0;
      A     L 1.1;
      JNB   _080;
      L     "coordinate".CoordinateCam_PP19[1].X;
      T     "DBWork".PointCamCheck[1].x;
_080: NOP   0;
      A     L 1.1;
      JNB   _081;
      L     "coordinate".CoordinateCam_PP19[1].Y;
      T     "DBWork".PointCamCheck[1].y;
_081: NOP   0;
      A     L 1.1;
      JNB   _082;
      L     "coordinate".TimeWeldingPP19[1];
      T     "DBWork".TempoSaldatura[1];
_082: NOP   0;
      A     L 1.1;
      JNB   _083;
      L     "coordinate".TimeWeldingPP19[2];
      T     "DBWork".TempoSaldatura[2];
_083: NOP   0;
      A     L 1.0;
      A     "On";
      A(;
      L     "Timer".NumberVane;
      L     20;
      ==I;
      );
      =     L 1.1;
      A     L 1.1;
      JNB   _084;
      CALL  "BLKMOV" (
           SRCBLK                   := "coordinate".CoordSaldaturaPP20,
           RET_VAL                  := MW 2044,
           DSTBLK                   := "DBWork".CoordSaldatura);
_084: NOP   0;
      A     L 1.1;
      JNB   _085;
      L     "coordinate".NumeroSaldaturePP20;
      T     "DBWork".NumeroSaldature;
_085: NOP   0;
      A     L 1.1;
      JNB   _086;
      L     "coordinate".CoordinateCam_PP20[1].X;
      T     "DBWork".PointCamCheck[1].x;
_086: NOP   0;
      A     L 1.1;
      JNB   _087;
      L     "coordinate".CoordinateCam_PP20[1].Y;
      T     "DBWork".PointCamCheck[1].y;
_087: NOP   0;
      A     L 1.1;
      JNB   _088;
      L     "coordinate".TimeWeldingPP20[1];
      T     "DBWork".TempoSaldatura[1];
_088: NOP   0;
      A     L 1.1;
      JNB   _089;
      L     "coordinate".TimeWeldingPP20[2];
      T     "DBWork".TempoSaldatura[2];
_089: NOP   0;
NETWORK
TITLE =
NETWORK
TITLE = TeachIn finish, save value for PP1
//Salvo sul Db Coordinate  i nuovi valori impostati con il teachIn per PP1.
      A     "Type_PP1";
      A     "M75.1";
      =     L 1.0;
      A     L 1.0;
      A     "On";
      A(;
      L     "Timer".NumberVane;
      L     1;
      ==I;
      );
      =     L 1.1;
      A     L 1.1;
      JNB   _08a;
      CALL  "BLKMOV" (
           SRCBLK                   := "DBWork".CoordSaldatura,
           RET_VAL                  := MW 2044,
           DSTBLK                   := "coordinate".CoordSaldaturaPP1);
_08a: A     BR;
      R     "M75.1";
      A     L 1.1;
      JNB   _08b;
      L     "DBWork".PointCamCheck[1].x;
      T     "coordinate".CoordinateCam_PP1[1].X;
_08b: NOP   0;
      A     L 1.1;
      JNB   _08c;
      L     "DBWork".PointCamCheck[1].y;
      T     "coordinate".CoordinateCam_PP1[1].Y;
_08c: NOP   0;
      A     L 1.0;
      A     "On";
      A(;
      L     "Timer".NumberVane;
      L     2;
      ==I;
      );
      =     L 1.1;
      A     L 1.1;
      JNB   _08d;
      CALL  "BLKMOV" (
           SRCBLK                   := "DBWork".CoordSaldatura,
           RET_VAL                  := MW 2044,
           DSTBLK                   := "coordinate".CoordSaldaturaPP2);
_08d: A     BR;
      R     "M75.1";
      A     L 1.1;
      JNB   _08e;
      L     "DBWork".PointCamCheck[1].x;
      T     "coordinate".CoordinateCam_PP2[1].X;
_08e: NOP   0;
      A     L 1.1;
      JNB   _08f;
      L     "DBWork".PointCamCheck[1].y;
      T     "coordinate".CoordinateCam_PP2[1].Y;
_08f: NOP   0;
      A     L 1.0;
      A     "On";
      A(;
      L     "Timer".NumberVane;
      L     3;
      ==I;
      );
      =     L 1.1;
      A     L 1.1;
      JNB   _090;
      CALL  "BLKMOV" (
           SRCBLK                   := "DBWork".CoordSaldatura,
           RET_VAL                  := MW 2044,
           DSTBLK                   := "coordinate".CoordSaldaturaPP3);
_090: A     BR;
      R     "M75.1";
      A     L 1.1;
      JNB   _091;
      L     "DBWork".PointCamCheck[1].x;
      T     "coordinate".CoordinateCam_PP3[1].X;
_091: NOP   0;
      A     L 1.1;
      JNB   _092;
      L     "DBWork".PointCamCheck[1].y;
      T     "coordinate".CoordinateCam_PP3[1].Y;
_092: NOP   0;
      A     L 1.0;
      A     "On";
      A(;
      L     "Timer".NumberVane;
      L     4;
      ==I;
      );
      =     L 1.1;
      A     L 1.1;
      JNB   _093;
      CALL  "BLKMOV" (
           SRCBLK                   := "DBWork".CoordSaldatura,
           RET_VAL                  := MW 2044,
           DSTBLK                   := "coordinate".CoordSaldaturaPP4);
_093: A     BR;
      R     "M75.1";
      A     L 1.1;
      JNB   _094;
      L     "DBWork".PointCamCheck[1].x;
      T     "coordinate".CoordinateCam_PP4[1].X;
_094: NOP   0;
      A     L 1.1;
      JNB   _095;
      L     "DBWork".PointCamCheck[1].y;
      T     "coordinate".CoordinateCam_PP4[1].Y;
_095: NOP   0;
      A     L 1.0;
      A     "On";
      A(;
      L     "Timer".NumberVane;
      L     5;
      ==I;
      );
      =     L 1.1;
      A     L 1.1;
      JNB   _096;
      CALL  "BLKMOV" (
           SRCBLK                   := "DBWork".CoordSaldatura,
           RET_VAL                  := MW 2044,
           DSTBLK                   := "coordinate".CoordSaldaturaPP5);
_096: A     BR;
      R     "M75.1";
      A     L 1.1;
      JNB   _097;
      L     "DBWork".PointCamCheck[1].x;
      T     "coordinate".CoordinateCam_PP5[1].X;
_097: NOP   0;
      A     L 1.1;
      JNB   _098;
      L     "DBWork".PointCamCheck[1].y;
      T     "coordinate".CoordinateCam_PP5[1].Y;
_098: NOP   0;
NETWORK
TITLE = TeachIn finish, save value for PP2
//Salvo sul Db Coordinate  i nuovi valori impostati con il teachIn per PP2.
      A     "Type_PP2";
      A     "M75.1";
      =     L 1.0;
      A     L 1.0;
      A     "On";
      A(;
      L     "Timer".NumberVane;
      L     6;
      ==I;
      );
      =     L 1.1;
      A     L 1.1;
      JNB   _099;
      CALL  "BLKMOV" (
           SRCBLK                   := "DBWork".CoordSaldatura,
           RET_VAL                  := MW 2044,
           DSTBLK                   := "coordinate".CoordSaldaturaPP6);
_099: A     BR;
      R     "M75.1";
      A     L 1.1;
      JNB   _09a;
      L     "DBWork".PointCamCheck[1].x;
      T     "coordinate".CoordinateCam_PP6[1].X;
_09a: NOP   0;
      A     L 1.1;
      JNB   _09b;
      L     "DBWork".PointCamCheck[1].y;
      T     "coordinate".CoordinateCam_PP6[1].Y;
_09b: NOP   0;
      A     L 1.0;
      A     "On";
      A(;
      L     "Timer".NumberVane;
      L     7;
      ==I;
      );
      =     L 1.1;
      A     L 1.1;
      JNB   _09c;
      CALL  "BLKMOV" (
           SRCBLK                   := "DBWork".CoordSaldatura,
           RET_VAL                  := MW 2044,
           DSTBLK                   := "coordinate".CoordSaldaturaPP7);
_09c: A     BR;
      R     "M75.1";
      A     L 1.1;
      JNB   _09d;
      L     "DBWork".PointCamCheck[1].x;
      T     "coordinate".CoordinateCam_PP7[1].X;
_09d: NOP   0;
      A     L 1.1;
      JNB   _09e;
      L     "DBWork".PointCamCheck[1].y;
      T     "coordinate".CoordinateCam_PP7[1].Y;
_09e: NOP   0;
      A     L 1.0;
      A     "On";
      A(;
      L     "Timer".NumberVane;
      L     8;
      ==I;
      );
      =     L 1.1;
      A     L 1.1;
      JNB   _09f;
      CALL  "BLKMOV" (
           SRCBLK                   := "DBWork".CoordSaldatura,
           RET_VAL                  := MW 2044,
           DSTBLK                   := "coordinate".CoordSaldaturaPP8);
_09f: A     BR;
      R     "M75.1";
      A     L 1.1;
      JNB   _0a0;
      L     "DBWork".PointCamCheck[1].x;
      T     "coordinate".CoordinateCam_PP8[1].X;
_0a0: NOP   0;
      A     L 1.1;
      JNB   _0a1;
      L     "DBWork".PointCamCheck[1].y;
      T     "coordinate".CoordinateCam_PP8[1].Y;
_0a1: NOP   0;
      A     L 1.0;
      A     "On";
      A(;
      L     "Timer".NumberVane;
      L     9;
      ==I;
      );
      =     L 1.1;
      A     L 1.1;
      JNB   _0a2;
      CALL  "BLKMOV" (
           SRCBLK                   := "DBWork".CoordSaldatura,
           RET_VAL                  := MW 2044,
           DSTBLK                   := "coordinate".CoordSaldaturaPP9);
_0a2: A     BR;
      R     "M75.1";
      A     L 1.1;
      JNB   _0a3;
      L     "DBWork".PointCamCheck[1].x;
      T     "coordinate".CoordinateCam_PP9[1].X;
_0a3: NOP   0;
      A     L 1.1;
      JNB   _0a4;
      L     "DBWork".PointCamCheck[1].y;
      T     "coordinate".CoordinateCam_PP9[1].Y;
_0a4: NOP   0;
      A     L 1.0;
      A     "On";
      A(;
      L     "Timer".NumberVane;
      L     10;
      ==I;
      );
      =     L 1.1;
      A     L 1.1;
      JNB   _0a5;
      CALL  "BLKMOV" (
           SRCBLK                   := "DBWork".CoordSaldatura,
           RET_VAL                  := MW 2044,
           DSTBLK                   := "coordinate".CoordSaldaturaPP10);
_0a5: A     BR;
      R     "M75.1";
      A     L 1.1;
      JNB   _0a6;
      L     "DBWork".PointCamCheck[1].x;
      T     "coordinate".CoordinateCam_PP10[1].X;
_0a6: NOP   0;
      A     L 1.1;
      JNB   _0a7;
      L     "DBWork".PointCamCheck[1].y;
      T     "coordinate".CoordinateCam_PP10[1].Y;
_0a7: NOP   0;
NETWORK
TITLE = TeachIn finish, save value for PP3
//Salvo sul Db Coordinate  i nuovi valori impostati con il teachIn per PP3.
      A     "Type_PP3";
      A     "M75.1";
      =     L 1.0;
      A     L 1.0;
      A     "On";
      A(;
      L     "Timer".NumberVane;
      L     11;
      ==I;
      );
      =     L 1.1;
      A     L 1.1;
      JNB   _0a8;
      CALL  "BLKMOV" (
           SRCBLK                   := "DBWork".CoordSaldatura,
           RET_VAL                  := MW 2044,
           DSTBLK                   := "coordinate".CoordSaldaturaPP11);
_0a8: A     BR;
      R     "M75.1";
      A     L 1.1;
      JNB   _0a9;
      L     "DBWork".PointCamCheck[1].x;
      T     "coordinate".CoordinateCam_PP11[1].X;
_0a9: NOP   0;
      A     L 1.1;
      JNB   _0aa;
      L     "DBWork".PointCamCheck[1].y;
      T     "coordinate".CoordinateCam_PP11[1].Y;
_0aa: NOP   0;
      A     L 1.0;
      A     "On";
      A(;
      L     "Timer".NumberVane;
      L     12;
      ==I;
      );
      =     L 1.1;
      A     L 1.1;
      JNB   _0ab;
      CALL  "BLKMOV" (
           SRCBLK                   := "DBWork".CoordSaldatura,
           RET_VAL                  := MW 2044,
           DSTBLK                   := "coordinate".CoordSaldaturaPP12);
_0ab: A     BR;
      R     "M75.1";
      A     L 1.1;
      JNB   _0ac;
      L     "DBWork".PointCamCheck[1].x;
      T     "coordinate".CoordinateCam_PP12[1].X;
_0ac: NOP   0;
      A     L 1.1;
      JNB   _0ad;
      L     "DBWork".PointCamCheck[1].y;
      T     "coordinate".CoordinateCam_PP12[1].Y;
_0ad: NOP   0;
      A     L 1.0;
      A     "On";
      A(;
      L     "Timer".NumberVane;
      L     13;
      ==I;
      );
      =     L 1.1;
      A     L 1.1;
      JNB   _0ae;
      CALL  "BLKMOV" (
           SRCBLK                   := "DBWork".CoordSaldatura,
           RET_VAL                  := MW 2044,
           DSTBLK                   := "coordinate".CoordSaldaturaPP13);
_0ae: A     BR;
      R     "M75.1";
      A     L 1.1;
      JNB   _0af;
      L     "DBWork".PointCamCheck[1].x;
      T     "coordinate".CoordinateCam_PP13[1].X;
_0af: NOP   0;
      A     L 1.1;
      JNB   _0b0;
      L     "DBWork".PointCamCheck[1].y;
      T     "coordinate".CoordinateCam_PP13[1].Y;
_0b0: NOP   0;
      A     L 1.0;
      A     "On";
      A(;
      L     "Timer".NumberVane;
      L     14;
      ==I;
      );
      =     L 1.1;
      A     L 1.1;
      JNB   _0b1;
      CALL  "BLKMOV" (
           SRCBLK                   := "DBWork".CoordSaldatura,
           RET_VAL                  := MW 2044,
           DSTBLK                   := "coordinate".CoordSaldaturaPP14);
_0b1: A     BR;
      R     "M75.1";
      A     L 1.1;
      JNB   _0b2;
      L     "DBWork".PointCamCheck[1].x;
      T     "coordinate".CoordinateCam_PP14[1].X;
_0b2: NOP   0;
      A     L 1.1;
      JNB   _0b3;
      L     "DBWork".PointCamCheck[1].y;
      T     "coordinate".CoordinateCam_PP14[1].Y;
_0b3: NOP   0;
      A     L 1.0;
      A     "On";
      A(;
      L     "Timer".NumberVane;
      L     15;
      ==I;
      );
      =     L 1.1;
      A     L 1.1;
      JNB   _0b4;
      CALL  "BLKMOV" (
           SRCBLK                   := "DBWork".CoordSaldatura,
           RET_VAL                  := MW 2044,
           DSTBLK                   := "coordinate".CoordSaldaturaPP15);
_0b4: A     BR;
      R     "M75.1";
      A     L 1.1;
      JNB   _0b5;
      L     "DBWork".PointCamCheck[1].x;
      T     "coordinate".CoordinateCam_PP15[1].X;
_0b5: NOP   0;
      A     L 1.1;
      JNB   _0b6;
      L     "DBWork".PointCamCheck[1].y;
      T     "coordinate".CoordinateCam_PP15[1].Y;
_0b6: NOP   0;
NETWORK
TITLE = TeachIn finish, save value for PP4
//Salvo sul Db Coordinate  i nuovi valori impostati con il teachIn per PP4.
      A     "Type_PP4";
      A     "M75.1";
      =     L 1.0;
      A     L 1.0;
      A     "On";
      A(;
      L     "Timer".NumberVane;
      L     16;
      ==I;
      );
      =     L 1.1;
      A     L 1.1;
      JNB   _0b7;
      CALL  "BLKMOV" (
           SRCBLK                   := "DBWork".CoordSaldatura,
           RET_VAL                  := MW 2044,
           DSTBLK                   := "coordinate".CoordSaldaturaPP16);
_0b7: A     BR;
      R     "M75.1";
      A     L 1.1;
      JNB   _0b8;
      L     "DBWork".PointCamCheck[1].x;
      T     "coordinate".CoordinateCam_PP16[1].X;
_0b8: NOP   0;
      A     L 1.1;
      JNB   _0b9;
      L     "DBWork".PointCamCheck[1].y;
      T     "coordinate".CoordinateCam_PP16[1].Y;
_0b9: NOP   0;
      A     L 1.0;
      A     "On";
      A(;
      L     "Timer".NumberVane;
      L     17;
      ==I;
      );
      =     L 1.1;
      A     L 1.1;
      JNB   _0ba;
      CALL  "BLKMOV" (
           SRCBLK                   := "DBWork".CoordSaldatura,
           RET_VAL                  := MW 2044,
           DSTBLK                   := "coordinate".CoordSaldaturaPP17);
_0ba: A     BR;
      R     "M75.1";
      A     L 1.1;
      JNB   _0bb;
      L     "DBWork".PointCamCheck[1].x;
      T     "coordinate".CoordinateCam_PP17[1].X;
_0bb: NOP   0;
      A     L 1.1;
      JNB   _0bc;
      L     "DBWork".PointCamCheck[1].y;
      T     "coordinate".CoordinateCam_PP17[1].Y;
_0bc: NOP   0;
      A     L 1.0;
      A     "On";
      A(;
      L     "Timer".NumberVane;
      L     18;
      ==I;
      );
      =     L 1.1;
      A     L 1.1;
      JNB   _0bd;
      CALL  "BLKMOV" (
           SRCBLK                   := "DBWork".CoordSaldatura,
           RET_VAL                  := MW 2044,
           DSTBLK                   := "coordinate".CoordSaldaturaPP18);
_0bd: A     BR;
      R     "M75.1";
      A     L 1.1;
      JNB   _0be;
      L     "DBWork".PointCamCheck[1].x;
      T     "coordinate".CoordinateCam_PP18[1].X;
_0be: NOP   0;
      A     L 1.1;
      JNB   _0bf;
      L     "DBWork".PointCamCheck[1].y;
      T     "coordinate".CoordinateCam_PP18[1].Y;
_0bf: NOP   0;
      A     L 1.0;
      A     "On";
      A(;
      L     "Timer".NumberVane;
      L     19;
      ==I;
      );
      =     L 1.1;
      A     L 1.1;
      JNB   _0c0;
      CALL  "BLKMOV" (
           SRCBLK                   := "DBWork".CoordSaldatura,
           RET_VAL                  := MW 2044,
           DSTBLK                   := "coordinate".CoordSaldaturaPP19);
_0c0: A     BR;
      R     "M75.1";
      A     L 1.1;
      JNB   _0c1;
      L     "DBWork".PointCamCheck[1].x;
      T     "coordinate".CoordinateCam_PP19[1].X;
_0c1: NOP   0;
      A     L 1.1;
      JNB   _0c2;
      L     "DBWork".PointCamCheck[1].y;
      T     "coordinate".CoordinateCam_PP19[1].Y;
_0c2: NOP   0;
      A     L 1.0;
      A     "On";
      A(;
      L     "Timer".NumberVane;
      L     20;
      ==I;
      );
      =     L 1.1;
      A     L 1.1;
      JNB   _0c3;
      CALL  "BLKMOV" (
           SRCBLK                   := "DBWork".CoordSaldatura,
           RET_VAL                  := MW 2044,
           DSTBLK                   := "coordinate".CoordSaldaturaPP20);
_0c3: A     BR;
      R     "M75.1";
      A     L 1.1;
      JNB   _0c4;
      L     "DBWork".PointCamCheck[1].x;
      T     "coordinate".CoordinateCam_PP20[1].X;
_0c4: NOP   0;
      A     L 1.1;
      JNB   _0c5;
      L     "DBWork".PointCamCheck[1].y;
      T     "coordinate".CoordinateCam_PP20[1].Y;
_0c5: NOP   0;
NETWORK
TITLE = Nozzle Components Ok
      A(;
      A     "Type_PP1";
      A     "M14.0";
      A     "M14.1";
      A     "M14.2";
      A     "M14.3";
      A     "M14.4";
      A     "M14.5";
      A     "M14.6";
      A     "M14.7";
      A     "M15.0";
      A     "M15.1";
      A     "M15.4";
      O;
      A     "Type_PP3";
      A     "M14.0";
      A     "M14.1";
      A     "M14.2";
      A     "M14.3";
      A     "M14.4";
      A     "M14.5";
      A     "M14.6";
      A     "M14.7";
      A     "M15.0";
      A     "M15.1";
      A     "M15.2";
      A(;
      O     "M15.3";
      O     "On";
      );
      A     "M15.4";
      A     "M15.5";
      O;
      A     "Type_PP2";
      A     "M14.0";
      A     "M14.1";
      A     "M14.2";
      A     "M14.3";
      A     "M14.4";
      A     "M14.5";
      A     "M14.6";
      A     "M14.7";
      A     "M15.0";
      A     "M15.1";
      A     "M15.2";
      A     "M15.4";
      O;
      A     "Type_PP4";
      A     "M14.0";
      A     "M14.1";
      A     "M14.2";
      A     "M14.3";
      A     "M14.4";
      A     "M14.5";
      A     "M14.6";
      A     "M14.7";
      A     "M15.0";
      A     "M15.1";
      A     "M15.2";
      A     "M15.3";
      A     "M15.4";
      A(;
      O     "M15.5";
      O     "On";
      );
      );
      A     "On";
      =     "M70.0";
NETWORK
TITLE = Save value for time
      A     "M11.2";
      A(;
      L     "DatiOP170B".NumeroPagina.NumeroPaginaCorrente;
      L     10;
      ==I;
      );
      A     "M2034.7";
      =     L 1.0;
      A     L 1.0;
      A     "Type_PP1";
      =     L 1.1;
      A     L 1.1;
      A(;
      L     "Timer".NumberVane;
      L     1;
      ==I;
      );
      =     L 1.2;
      A     L 1.2;
      JNB   _0c6;
      L     "DBWork".TempoSaldatura[1];
      T     "coordinate".TimeWeldingPP1[1];
_0c6: NOP   0;
      A     L 1.2;
      JNB   _0c7;
      L     "DBWork".TempoSaldatura[2];
      T     "coordinate".TimeWeldingPP1[2];
_0c7: NOP   0;
      A     L 1.1;
      A(;
      L     "Timer".NumberVane;
      L     2;
      ==I;
      );
      =     L 1.2;
      A     L 1.2;
      JNB   _0c8;
      L     "DBWork".TempoSaldatura[1];
      T     "coordinate".TimeWeldingPP2[1];
_0c8: NOP   0;
      A     L 1.2;
      JNB   _0c9;
      L     "DBWork".TempoSaldatura[2];
      T     "coordinate".TimeWeldingPP2[2];
_0c9: NOP   0;
      A     L 1.1;
      A(;
      L     "Timer".NumberVane;
      L     3;
      ==I;
      );
      =     L 1.2;
      A     L 1.2;
      JNB   _0ca;
      L     "DBWork".TempoSaldatura[1];
      T     "coordinate".TimeWeldingPP3[1];
_0ca: NOP   0;
      A     L 1.2;
      JNB   _0cb;
      L     "DBWork".TempoSaldatura[2];
      T     "coordinate".TimeWeldingPP3[2];
_0cb: NOP   0;
      A     L 1.1;
      A(;
      L     "Timer".NumberVane;
      L     4;
      ==I;
      );
      =     L 1.2;
      A     L 1.2;
      JNB   _0cc;
      L     "DBWork".TempoSaldatura[1];
      T     "coordinate".TimeWeldingPP4[1];
_0cc: NOP   0;
      A     L 1.2;
      JNB   _0cd;
      L     "DBWork".TempoSaldatura[2];
      T     "coordinate".TimeWeldingPP4[2];
_0cd: NOP   0;
      A     L 1.1;
      A(;
      L     "Timer".NumberVane;
      L     5;
      ==I;
      );
      =     L 1.2;
      A     L 1.2;
      JNB   _0ce;
      L     "DBWork".TempoSaldatura[1];
      T     "coordinate".TimeWeldingPP5[1];
_0ce: NOP   0;
      A     L 1.2;
      JNB   _0cf;
      L     "DBWork".TempoSaldatura[2];
      T     "coordinate".TimeWeldingPP5[2];
_0cf: NOP   0;
      A     L 1.0;
      A     "Type_PP2";
      =     L 1.1;
      A     L 1.1;
      A(;
      L     "Timer".NumberVane;
      L     6;
      ==I;
      );
      =     L 1.2;
      A     L 1.2;
      JNB   _0d0;
      L     "DBWork".TempoSaldatura[1];
      T     "coordinate".TimeWeldingPP6[1];
_0d0: NOP   0;
      A     L 1.2;
      JNB   _0d1;
      L     "DBWork".TempoSaldatura[2];
      T     "coordinate".TimeWeldingPP6[2];
_0d1: NOP   0;
      A     L 1.1;
      A(;
      L     "Timer".NumberVane;
      L     7;
      ==I;
      );
      =     L 1.2;
      A     L 1.2;
      JNB   _0d2;
      L     "DBWork".TempoSaldatura[1];
      T     "coordinate".TimeWeldingPP7[1];
_0d2: NOP   0;
      A     L 1.2;
      JNB   _0d3;
      L     "DBWork".TempoSaldatura[2];
      T     "coordinate".TimeWeldingPP7[2];
_0d3: NOP   0;
      A     L 1.1;
      A(;
      L     "Timer".NumberVane;
      L     8;
      ==I;
      );
      =     L 1.2;
      A     L 1.2;
      JNB   _0d4;
      L     "DBWork".TempoSaldatura[1];
      T     "coordinate".TimeWeldingPP8[1];
_0d4: NOP   0;
      A     L 1.2;
      JNB   _0d5;
      L     "DBWork".TempoSaldatura[2];
      T     "coordinate".TimeWeldingPP8[2];
_0d5: NOP   0;
      A     L 1.1;
      A(;
      L     "Timer".NumberVane;
      L     9;
      ==I;
      );
      =     L 1.2;
      A     L 1.2;
      JNB   _0d6;
      L     "DBWork".TempoSaldatura[1];
      T     "coordinate".TimeWeldingPP9[1];
_0d6: NOP   0;
      A     L 1.2;
      JNB   _0d7;
      L     "DBWork".TempoSaldatura[2];
      T     "coordinate".TimeWeldingPP9[2];
_0d7: NOP   0;
      A     L 1.1;
      A(;
      L     "Timer".NumberVane;
      L     10;
      ==I;
      );
      =     L 1.2;
      A     L 1.2;
      JNB   _0d8;
      L     "DBWork".TempoSaldatura[1];
      T     "coordinate".TimeWeldingPP10[1];
_0d8: NOP   0;
      A     L 1.2;
      JNB   _0d9;
      L     "DBWork".TempoSaldatura[2];
      T     "coordinate".TimeWeldingPP10[2];
_0d9: NOP   0;
      A     L 1.0;
      A     "Type_PP3";
      A(;
      L     "Timer".NumberVane;
      L     11;
      ==I;
      );
      =     L 1.1;
      A     L 1.1;
      JNB   _0da;
      L     "DBWork".TempoSaldatura[1];
      T     "coordinate".TimeWeldingPP3[1];
_0da: NOP   0;
      A     L 1.1;
      JNB   _0db;
      L     "DBWork".TempoSaldatura[2];
      T     "coordinate".TimeWeldingPP3[2];
_0db: NOP   0;
      A     L 1.0;
      A     "Type_PP4";
      =     L 1.1;
      A     L 1.1;
      A(;
      L     "Timer".NumberVane;
      L     16;
      ==I;
      );
      =     L 1.2;
      A     L 1.2;
      JNB   _0dc;
      L     "DBWork".TempoSaldatura[1];
      T     "coordinate".TimeWeldingPP16[1];
_0dc: NOP   0;
      A     L 1.2;
      JNB   _0dd;
      L     "DBWork".TempoSaldatura[2];
      T     "coordinate".TimeWeldingPP16[2];
_0dd: NOP   0;
      A     L 1.1;
      A(;
      L     "Timer".NumberVane;
      L     17;
      ==I;
      );
      =     L 1.2;
      A     L 1.2;
      JNB   _0de;
      L     "DBWork".TempoSaldatura[1];
      T     "coordinate".TimeWeldingPP17[1];
_0de: NOP   0;
      A     L 1.2;
      JNB   _0df;
      L     "DBWork".TempoSaldatura[2];
      T     "coordinate".TimeWeldingPP17[2];
_0df: NOP   0;
      A     L 1.1;
      A(;
      L     "Timer".NumberVane;
      L     18;
      ==I;
      );
      =     L 1.2;
      A     L 1.2;
      JNB   _0e0;
      L     "DBWork".TempoSaldatura[1];
      T     "coordinate".TimeWeldingPP18[1];
_0e0: NOP   0;
      A     L 1.2;
      JNB   _0e1;
      L     "DBWork".TempoSaldatura[2];
      T     "coordinate".TimeWeldingPP18[2];
_0e1: NOP   0;
      A     L 1.1;
      A(;
      L     "Timer".NumberVane;
      L     19;
      ==I;
      );
      =     L 1.2;
      A     L 1.2;
      JNB   _0e2;
      L     "DBWork".TempoSaldatura[1];
      T     "coordinate".TimeWeldingPP19[1];
_0e2: NOP   0;
      A     L 1.2;
      JNB   _0e3;
      L     "DBWork".TempoSaldatura[2];
      T     "coordinate".TimeWeldingPP19[2];
_0e3: NOP   0;
      A     L 1.1;
      A(;
      L     "Timer".NumberVane;
      L     20;
      ==I;
      );
      =     L 1.2;
      A     L 1.2;
      JNB   _0e4;
      L     "DBWork".TempoSaldatura[1];
      T     "coordinate".TimeWeldingPP20[1];
_0e4: NOP   0;
      A     L 1.2;
      JNB   _0e5;
      L     "DBWork".TempoSaldatura[2];
      T     "coordinate".TimeWeldingPP20[2];
_0e5: NOP   0;
NETWORK
TITLE =
NETWORK
TITLE = load value for selected point, use it in auto, teach in and weld
//carico le coordinate del punto selezionato per fare le saldature in automatico 
//per il teachIn e per il test di salsatura
      A     "On";
      =     L 0.0;
      A     L 0.0;
      A(;
      A(;
      L     "DBWork".PP[1].NumSaldaturaAtt;
      L     0;
      ==I;
      );
      A     "AUT";
      O;
      A     "M11.2";
      A(;
      L     "DatiOP170B".PointWeldingTeachIn;
      L     1;
      ==I;
      );
      A(;
      O(;
      L     "DatiOP170B".NumeroPagina.NumeroPaginaCorrente;
      L     5;
      ==I;
      );
      O(;
      L     "DatiOP170B".NumeroPagina.NumeroPaginaCorrente;
      L     11;
      ==I;
      );
      );
      );
      =     L 0.1;
      A(;
      A     L 0.1;
      A     "DBWork".RotationTable;
      JNB   _0e6;
      L     "DBWork".CoordSaldatura[1].X1;
      T     "MD588";
      SET;
      SAVE;
      CLR;
_0e6: A     BR;
      );
      JNB   _0e7;
      L     "DBWork".CoordSaldatura[1].Y1;
      T     "MD592";
_0e7: NOP   0;
      A(;
      A     L 0.1;
      AN    "DBWork".RotationTable;
      JNB   _0e8;
      L     "DBWork".CoordSaldatura[1].X2;
      T     "MD588";
      SET;
      SAVE;
      CLR;
_0e8: A     BR;
      );
      JNB   _0e9;
      L     "DBWork".CoordSaldatura[1].Y2;
      T     "MD592";
_0e9: NOP   0;
      A     L 0.0;
      A(;
      A(;
      L     "DBWork".PP[1].NumSaldaturaAtt;
      L     1;
      ==I;
      );
      A     "AUT";
      O;
      A     "M11.2";
      A(;
      L     "DatiOP170B".PointWeldingTeachIn;
      L     2;
      ==I;
      );
      A(;
      O(;
      L     "DatiOP170B".NumeroPagina.NumeroPaginaCorrente;
      L     5;
      ==I;
      );
      O(;
      L     "DatiOP170B".NumeroPagina.NumeroPaginaCorrente;
      L     11;
      ==I;
      );
      );
      );
      =     L 0.1;
      A(;
      A     L 0.1;
      A     "DBWork".RotationTable;
      JNB   _0ea;
      L     "DBWork".CoordSaldatura[2].X1;
      T     "MD588";
      SET;
      SAVE;
      CLR;
_0ea: A     BR;
      );
      JNB   _0eb;
      L     "DBWork".CoordSaldatura[2].Y1;
      T     "MD592";
_0eb: NOP   0;
      A(;
      A     L 0.1;
      AN    "DBWork".RotationTable;
      JNB   _0ec;
      L     "DBWork".CoordSaldatura[2].X2;
      T     "MD588";
      SET;
      SAVE;
      CLR;
_0ec: A     BR;
      );
      JNB   _0ed;
      L     "DBWork".CoordSaldatura[2].Y2;
      T     "MD592";
_0ed: NOP   0;
      A     L 0.0;
      A(;
      A(;
      L     "DBWork".PP[1].NumSaldaturaAtt;
      L     2;
      ==I;
      );
      A     "AUT";
      O;
      A     "M11.2";
      A(;
      L     "DatiOP170B".PointWeldingTeachIn;
      L     3;
      ==I;
      );
      A(;
      O(;
      L     "DatiOP170B".NumeroPagina.NumeroPaginaCorrente;
      L     5;
      ==I;
      );
      O(;
      L     "DatiOP170B".NumeroPagina.NumeroPaginaCorrente;
      L     11;
      ==I;
      );
      );
      );
      =     L 0.1;
      A(;
      A     L 0.1;
      A     "DBWork".RotationTable;
      JNB   _0ee;
      L     "DBWork".CoordSaldatura[3].X1;
      T     "MD588";
      SET;
      SAVE;
      CLR;
_0ee: A     BR;
      );
      JNB   _0ef;
      L     "DBWork".CoordSaldatura[3].Y1;
      T     "MD592";
_0ef: NOP   0;
      A(;
      A     L 0.1;
      AN    "DBWork".RotationTable;
      JNB   _0f0;
      L     "DBWork".CoordSaldatura[3].X2;
      T     "MD588";
      SET;
      SAVE;
      CLR;
_0f0: A     BR;
      );
      JNB   _0f1;
      L     "DBWork".CoordSaldatura[3].Y2;
      T     "MD592";
_0f1: NOP   0;
      A     L 0.0;
      A(;
      A(;
      L     "DBWork".PP[1].NumSaldaturaAtt;
      L     3;
      ==I;
      );
      A     "AUT";
      O;
      A     "M11.2";
      A(;
      L     "DatiOP170B".PointWeldingTeachIn;
      L     4;
      ==I;
      );
      A(;
      O(;
      L     "DatiOP170B".NumeroPagina.NumeroPaginaCorrente;
      L     5;
      ==I;
      );
      O(;
      L     "DatiOP170B".NumeroPagina.NumeroPaginaCorrente;
      L     11;
      ==I;
      );
      );
      );
      =     L 0.1;
      A(;
      A     L 0.1;
      A     "DBWork".RotationTable;
      JNB   _0f2;
      L     "DBWork".CoordSaldatura[4].X1;
      T     "MD588";
      SET;
      SAVE;
      CLR;
_0f2: A     BR;
      );
      JNB   _0f3;
      L     "DBWork".CoordSaldatura[4].Y1;
      T     "MD592";
_0f3: NOP   0;
      A(;
      A     L 0.1;
      AN    "DBWork".RotationTable;
      JNB   _0f4;
      L     "DBWork".CoordSaldatura[4].X2;
      T     "MD588";
      SET;
      SAVE;
      CLR;
_0f4: A     BR;
      );
      JNB   _0f5;
      L     "DBWork".CoordSaldatura[4].Y2;
      T     "MD592";
_0f5: NOP   0;
      A     L 0.0;
      A(;
      A(;
      L     "DBWork".PP[1].NumSaldaturaAtt;
      L     4;
      ==I;
      );
      A     "AUT";
      O;
      A     "M11.2";
      A(;
      L     "DatiOP170B".PointWeldingTeachIn;
      L     5;
      ==I;
      );
      A(;
      O(;
      L     "DatiOP170B".NumeroPagina.NumeroPaginaCorrente;
      L     5;
      ==I;
      );
      O(;
      L     "DatiOP170B".NumeroPagina.NumeroPaginaCorrente;
      L     11;
      ==I;
      );
      );
      );
      =     L 0.1;
      A(;
      A     L 0.1;
      A     "DBWork".RotationTable;
      JNB   _0f6;
      L     "DBWork".CoordSaldatura[5].X1;
      T     "MD588";
      SET;
      SAVE;
      CLR;
_0f6: A     BR;
      );
      JNB   _0f7;
      L     "DBWork".CoordSaldatura[5].Y1;
      T     "MD592";
_0f7: NOP   0;
      A(;
      A     L 0.1;
      AN    "DBWork".RotationTable;
      JNB   _0f8;
      L     "DBWork".CoordSaldatura[5].X2;
      T     "MD588";
      SET;
      SAVE;
      CLR;
_0f8: A     BR;
      );
      JNB   _0f9;
      L     "DBWork".CoordSaldatura[5].Y2;
      T     "MD592";
_0f9: NOP   0;
      A     L 0.0;
      A(;
      A(;
      L     "DBWork".PP[1].NumSaldaturaAtt;
      L     5;
      ==I;
      );
      A     "AUT";
      O;
      A     "M11.2";
      A(;
      L     "DatiOP170B".PointWeldingTeachIn;
      L     6;
      ==I;
      );
      A(;
      O(;
      L     "DatiOP170B".NumeroPagina.NumeroPaginaCorrente;
      L     5;
      ==I;
      );
      O(;
      L     "DatiOP170B".NumeroPagina.NumeroPaginaCorrente;
      L     11;
      ==I;
      );
      );
      );
      =     L 0.1;
      A(;
      A     L 0.1;
      A     "DBWork".RotationTable;
      JNB   _0fa;
      L     "DBWork".CoordSaldatura[6].X1;
      T     "MD588";
      SET;
      SAVE;
      CLR;
_0fa: A     BR;
      );
      JNB   _0fb;
      L     "DBWork".CoordSaldatura[6].Y1;
      T     "MD592";
_0fb: NOP   0;
      A(;
      A     L 0.1;
      AN    "DBWork".RotationTable;
      JNB   _0fc;
      L     "DBWork".CoordSaldatura[6].X2;
      T     "MD588";
      SET;
      SAVE;
      CLR;
_0fc: A     BR;
      );
      JNB   _0fd;
      L     "DBWork".CoordSaldatura[6].Y2;
      T     "MD592";
_0fd: NOP   0;
      A     L 0.0;
      A(;
      A(;
      L     "DBWork".PP[1].NumSaldaturaAtt;
      L     6;
      ==I;
      );
      A     "AUT";
      O;
      A     "M11.2";
      A(;
      L     "DatiOP170B".PointWeldingTeachIn;
      L     7;
      ==I;
      );
      A(;
      O(;
      L     "DatiOP170B".NumeroPagina.NumeroPaginaCorrente;
      L     5;
      ==I;
      );
      O(;
      L     "DatiOP170B".NumeroPagina.NumeroPaginaCorrente;
      L     11;
      ==I;
      );
      );
      );
      =     L 0.1;
      A(;
      A     L 0.1;
      A     "DBWork".RotationTable;
      JNB   _0fe;
      L     "DBWork".CoordSaldatura[7].X1;
      T     "MD588";
      SET;
      SAVE;
      CLR;
_0fe: A     BR;
      );
      JNB   _0ff;
      L     "DBWork".CoordSaldatura[7].Y1;
      T     "MD592";
_0ff: NOP   0;
      A(;
      A     L 0.1;
      AN    "DBWork".RotationTable;
      JNB   _100;
      L     "DBWork".CoordSaldatura[7].X2;
      T     "MD588";
      SET;
      SAVE;
      CLR;
_100: A     BR;
      );
      JNB   _101;
      L     "DBWork".CoordSaldatura[7].Y2;
      T     "MD592";
_101: NOP   0;
      A     L 0.0;
      A(;
      A(;
      L     "DBWork".PP[1].NumSaldaturaAtt;
      L     7;
      ==I;
      );
      A     "AUT";
      O;
      A     "M11.2";
      A(;
      L     "DatiOP170B".PointWeldingTeachIn;
      L     8;
      ==I;
      );
      A(;
      O(;
      L     "DatiOP170B".NumeroPagina.NumeroPaginaCorrente;
      L     5;
      ==I;
      );
      O(;
      L     "DatiOP170B".NumeroPagina.NumeroPaginaCorrente;
      L     11;
      ==I;
      );
      );
      );
      =     L 0.1;
      A(;
      A     L 0.1;
      A     "DBWork".RotationTable;
      JNB   _102;
      L     "DBWork".CoordSaldatura[8].X1;
      T     "MD588";
      SET;
      SAVE;
      CLR;
_102: A     BR;
      );
      JNB   _103;
      L     "DBWork".CoordSaldatura[8].Y1;
      T     "MD592";
_103: NOP   0;
      A(;
      A     L 0.1;
      AN    "DBWork".RotationTable;
      JNB   _104;
      L     "DBWork".CoordSaldatura[8].X2;
      T     "MD588";
      SET;
      SAVE;
      CLR;
_104: A     BR;
      );
      JNB   _105;
      L     "DBWork".CoordSaldatura[8].Y2;
      T     "MD592";
_105: NOP   0;
      A     L 0.0;
      A(;
      A(;
      L     "DBWork".PP[1].NumSaldaturaAtt;
      L     8;
      ==I;
      );
      A     "AUT";
      O;
      A     "M11.2";
      A(;
      L     "DatiOP170B".PointWeldingTeachIn;
      L     9;
      ==I;
      );
      A(;
      O(;
      L     "DatiOP170B".NumeroPagina.NumeroPaginaCorrente;
      L     5;
      ==I;
      );
      O(;
      L     "DatiOP170B".NumeroPagina.NumeroPaginaCorrente;
      L     11;
      ==I;
      );
      );
      );
      =     L 0.1;
      A(;
      A     L 0.1;
      A     "DBWork".RotationTable;
      JNB   _106;
      L     "DBWork".CoordSaldatura[9].X1;
      T     "MD588";
      SET;
      SAVE;
      CLR;
_106: A     BR;
      );
      JNB   _107;
      L     "DBWork".CoordSaldatura[9].Y1;
      T     "MD592";
_107: NOP   0;
      A(;
      A     L 0.1;
      AN    "DBWork".RotationTable;
      JNB   _108;
      L     "DBWork".CoordSaldatura[9].X2;
      T     "MD588";
      SET;
      SAVE;
      CLR;
_108: A     BR;
      );
      JNB   _109;
      L     "DBWork".CoordSaldatura[9].Y2;
      T     "MD592";
_109: NOP   0;
      A     L 0.0;
      A(;
      A(;
      L     "DBWork".PP[1].NumSaldaturaAtt;
      L     9;
      ==I;
      );
      A     "AUT";
      O;
      A     "M11.2";
      A(;
      L     "DatiOP170B".PointWeldingTeachIn;
      L     10;
      ==I;
      );
      A(;
      O(;
      L     "DatiOP170B".NumeroPagina.NumeroPaginaCorrente;
      L     5;
      ==I;
      );
      O(;
      L     "DatiOP170B".NumeroPagina.NumeroPaginaCorrente;
      L     11;
      ==I;
      );
      );
      );
      =     L 0.1;
      A(;
      A     L 0.1;
      A     "DBWork".RotationTable;
      JNB   _10a;
      L     "DBWork".CoordSaldatura[10].X1;
      T     "MD588";
      SET;
      SAVE;
      CLR;
_10a: A     BR;
      );
      JNB   _10b;
      L     "DBWork".CoordSaldatura[10].Y1;
      T     "MD592";
_10b: NOP   0;
      A(;
      A     L 0.1;
      AN    "DBWork".RotationTable;
      JNB   _10c;
      L     "DBWork".CoordSaldatura[10].X2;
      T     "MD588";
      SET;
      SAVE;
      CLR;
_10c: A     BR;
      );
      JNB   _10d;
      L     "DBWork".CoordSaldatura[10].Y2;
      T     "MD592";
_10d: NOP   0;
      A     L 0.0;
      A(;
      A(;
      L     "DBWork".PP[1].NumSaldaturaAtt;
      L     10;
      ==I;
      );
      A     "AUT";
      O;
      A     "M11.2";
      A(;
      L     "DatiOP170B".PointWeldingTeachIn;
      L     11;
      ==I;
      );
      A(;
      O(;
      L     "DatiOP170B".NumeroPagina.NumeroPaginaCorrente;
      L     5;
      ==I;
      );
      O(;
      L     "DatiOP170B".NumeroPagina.NumeroPaginaCorrente;
      L     11;
      ==I;
      );
      );
      );
      =     L 0.1;
      A(;
      A     L 0.1;
      A     "DBWork".RotationTable;
      JNB   _10e;
      L     "DBWork".CoordSaldatura[11].X1;
      T     "MD588";
      SET;
      SAVE;
      CLR;
_10e: A     BR;
      );
      JNB   _10f;
      L     "DBWork".CoordSaldatura[11].Y1;
      T     "MD592";
_10f: NOP   0;
      A(;
      A     L 0.1;
      AN    "DBWork".RotationTable;
      JNB   _110;
      L     "DBWork".CoordSaldatura[11].X2;
      T     "MD588";
      SET;
      SAVE;
      CLR;
_110: A     BR;
      );
      JNB   _111;
      L     "DBWork".CoordSaldatura[11].Y2;
      T     "MD592";
_111: NOP   0;
      A     L 0.0;
      A(;
      A(;
      L     "DBWork".PP[1].NumSaldaturaAtt;
      L     11;
      ==I;
      );
      A     "AUT";
      O;
      A     "M11.2";
      A(;
      L     "DatiOP170B".PointWeldingTeachIn;
      L     12;
      ==I;
      );
      A(;
      O(;
      L     "DatiOP170B".NumeroPagina.NumeroPaginaCorrente;
      L     5;
      ==I;
      );
      O(;
      L     "DatiOP170B".NumeroPagina.NumeroPaginaCorrente;
      L     11;
      ==I;
      );
      );
      );
      =     L 0.1;
      A(;
      A     L 0.1;
      A     "DBWork".RotationTable;
      JNB   _112;
      L     "DBWork".CoordSaldatura[12].X1;
      T     "MD588";
      SET;
      SAVE;
      CLR;
_112: A     BR;
      );
      JNB   _113;
      L     "DBWork".CoordSaldatura[12].Y1;
      T     "MD592";
_113: NOP   0;
      A(;
      A     L 0.1;
      AN    "DBWork".RotationTable;
      JNB   _114;
      L     "DBWork".CoordSaldatura[12].X2;
      T     "MD588";
      SET;
      SAVE;
      CLR;
_114: A     BR;
      );
      JNB   _115;
      L     "DBWork".CoordSaldatura[12].Y2;
      T     "MD592";
_115: NOP   0;
      A     L 0.0;
      A(;
      A(;
      L     "DBWork".PP[1].NumSaldaturaAtt;
      L     12;
      ==I;
      );
      A     "AUT";
      O;
      A     "M11.2";
      A(;
      L     "DatiOP170B".PointWeldingTeachIn;
      L     13;
      ==I;
      );
      A(;
      O(;
      L     "DatiOP170B".NumeroPagina.NumeroPaginaCorrente;
      L     5;
      ==I;
      );
      O(;
      L     "DatiOP170B".NumeroPagina.NumeroPaginaCorrente;
      L     11;
      ==I;
      );
      );
      );
      =     L 0.1;
      A(;
      A     L 0.1;
      A     "DBWork".RotationTable;
      JNB   _116;
      L     "DBWork".CoordSaldatura[13].X1;
      T     "MD588";
      SET;
      SAVE;
      CLR;
_116: A     BR;
      );
      JNB   _117;
      L     "DBWork".CoordSaldatura[13].Y1;
      T     "MD592";
_117: NOP   0;
      A(;
      A     L 0.1;
      AN    "DBWork".RotationTable;
      JNB   _118;
      L     "DBWork".CoordSaldatura[13].X2;
      T     "MD588";
      SET;
      SAVE;
      CLR;
_118: A     BR;
      );
      JNB   _119;
      L     "DBWork".CoordSaldatura[13].Y2;
      T     "MD592";
_119: NOP   0;
NETWORK
TITLE = load value point for check with cam
//posizione per fare la foto
      A(;
      A     "On";
      A(;
      A(;
      O     "M61.0";
      O     "M22.0";
      );
      AN    "M61.1";
      A     "AUT";
      O;
      A     "M11.2";
      A(;
      L     "DatiOP170B".PointWeldingTeachIn;
      L     14;
      ==I;
      );
      A(;
      L     "DatiOP170B".NumeroPagina.NumeroPaginaCorrente;
      L     5;
      ==I;
      );
      );
      JNB   _11a;
      L     "DBWork".PointCamCheck[1].x;
      T     "MD588";
      SET;
      SAVE;
      CLR;
_11a: A     BR;
      );
      JNB   _11b;
      L     "DBWork".PointCamCheck[1].y;
      T     "MD592";
      SET;
      SAVE;
      CLR;
_11b: A     BR;
      S     "M63.6";
NETWORK
TITLE = ******************** Value point for Welding *******A***********
NETWORK
TITLE = i load value point respect type of tool A or B
//In base alla saldatura che effettuo passo le coordinate a gli assi
      A     "On";
      A     "AUT";
      A     "DBWork".RotationTable;
      =     L 1.0;
      A(;
      A     L 1.0;
      A(;
      L     "DBWork".PP[1].NumSaldaturaAtt;
      L     0;
      ==I;
      );
      JNB   _11c;
      L     "DBWork".CoordSaldatura[1].X1;
      T     "MD588";
      SET;
      SAVE;
      CLR;
_11c: A     BR;
      );
      JNB   _11d;
      L     "DBWork".CoordSaldatura[1].Y1;
      T     "MD592";
_11d: NOP   0;
      A(;
      A     L 1.0;
      A(;
      L     "DBWork".PP[1].NumSaldaturaAtt;
      L     1;
      ==I;
      );
      JNB   _11e;
      L     "DBWork".CoordSaldatura[2].X1;
      T     "MD588";
      SET;
      SAVE;
      CLR;
_11e: A     BR;
      );
      JNB   _11f;
      L     "DBWork".CoordSaldatura[2].Y1;
      T     "MD592";
_11f: NOP   0;
      A(;
      A     L 1.0;
      A(;
      L     "DBWork".PP[1].NumSaldaturaAtt;
      L     2;
      ==I;
      );
      JNB   _120;
      L     "DBWork".CoordSaldatura[3].X1;
      T     "MD588";
      SET;
      SAVE;
      CLR;
_120: A     BR;
      );
      JNB   _121;
      L     "DBWork".CoordSaldatura[3].Y1;
      T     "MD592";
_121: NOP   0;
      A(;
      A     L 1.0;
      A(;
      L     "DBWork".PP[1].NumSaldaturaAtt;
      L     3;
      ==I;
      );
      JNB   _122;
      L     "DBWork".CoordSaldatura[4].X1;
      T     "MD588";
      SET;
      SAVE;
      CLR;
_122: A     BR;
      );
      JNB   _123;
      L     "DBWork".CoordSaldatura[4].Y1;
      T     "MD592";
_123: NOP   0;
      A(;
      A     L 1.0;
      A(;
      L     "DBWork".PP[1].NumSaldaturaAtt;
      L     4;
      ==I;
      );
      JNB   _124;
      L     "DBWork".CoordSaldatura[5].X1;
      T     "MD588";
      SET;
      SAVE;
      CLR;
_124: A     BR;
      );
      JNB   _125;
      L     "DBWork".CoordSaldatura[5].Y1;
      T     "MD592";
_125: NOP   0;
      A(;
      A     L 1.0;
      A(;
      L     "DBWork".PP[1].NumSaldaturaAtt;
      L     5;
      ==I;
      );
      JNB   _126;
      L     "DBWork".CoordSaldatura[6].X1;
      T     "MD588";
      SET;
      SAVE;
      CLR;
_126: A     BR;
      );
      JNB   _127;
      L     "DBWork".CoordSaldatura[6].Y1;
      T     "MD592";
_127: NOP   0;
      A(;
      A     L 1.0;
      A(;
      L     "DBWork".PP[1].NumSaldaturaAtt;
      L     6;
      ==I;
      );
      JNB   _128;
      L     "DBWork".CoordSaldatura[7].X1;
      T     "MD588";
      SET;
      SAVE;
      CLR;
_128: A     BR;
      );
      JNB   _129;
      L     "DBWork".CoordSaldatura[7].Y1;
      T     "MD592";
_129: NOP   0;
      A(;
      A     L 1.0;
      A(;
      L     "DBWork".PP[1].NumSaldaturaAtt;
      L     7;
      ==I;
      );
      JNB   _12a;
      L     "DBWork".CoordSaldatura[8].X1;
      T     "MD588";
      SET;
      SAVE;
      CLR;
_12a: A     BR;
      );
      JNB   _12b;
      L     "DBWork".CoordSaldatura[8].Y1;
      T     "MD592";
_12b: NOP   0;
      A(;
      A     L 1.0;
      A(;
      L     "DBWork".PP[1].NumSaldaturaAtt;
      L     8;
      ==I;
      );
      JNB   _12c;
      L     "DBWork".CoordSaldatura[9].X1;
      T     "MD588";
      SET;
      SAVE;
      CLR;
_12c: A     BR;
      );
      JNB   _12d;
      L     "DBWork".CoordSaldatura[9].Y1;
      T     "MD592";
_12d: NOP   0;
      A(;
      A     L 1.0;
      A(;
      L     "DBWork".PP[1].NumSaldaturaAtt;
      L     9;
      ==I;
      );
      JNB   _12e;
      L     "DBWork".CoordSaldatura[10].X1;
      T     "MD588";
      SET;
      SAVE;
      CLR;
_12e: A     BR;
      );
      JNB   _12f;
      L     "DBWork".CoordSaldatura[10].Y1;
      T     "MD592";
_12f: NOP   0;
      A(;
      A     L 1.0;
      A(;
      L     "DBWork".PP[1].NumSaldaturaAtt;
      L     10;
      ==I;
      );
      JNB   _130;
      L     "DBWork".CoordSaldatura[11].X1;
      T     "MD588";
      SET;
      SAVE;
      CLR;
_130: A     BR;
      );
      JNB   _131;
      L     "DBWork".CoordSaldatura[11].Y1;
      T     "MD592";
_131: NOP   0;
      A(;
      A     L 1.0;
      A(;
      L     "DBWork".PP[1].NumSaldaturaAtt;
      L     11;
      ==I;
      );
      JNB   _132;
      L     "DBWork".CoordSaldatura[12].X1;
      T     "MD588";
      SET;
      SAVE;
      CLR;
_132: A     BR;
      );
      JNB   _133;
      L     "DBWork".CoordSaldatura[12].Y1;
      T     "MD592";
_133: NOP   0;
      A(;
      A     L 1.0;
      A(;
      L     "DBWork".PP[1].NumSaldaturaAtt;
      L     12;
      ==I;
      );
      JNB   _134;
      L     "DBWork".CoordSaldatura[13].X1;
      T     "MD588";
      SET;
      SAVE;
      CLR;
_134: A     BR;
      );
      JNB   _135;
      L     "DBWork".CoordSaldatura[13].Y1;
      T     "MD592";
_135: NOP   0;
NETWORK
TITLE = ******************** Value Point for Welding *********B********
NETWORK
TITLE = i load value point respect type of tool A or B
//In base alla saldatura che effettuo passo le coordinate a gli assi
      A     "On";
      A     "AUT";
      AN    "DBWork".RotationTable;
      =     L 1.0;
      A(;
      A     L 1.0;
      A(;
      L     "DBWork".PP[1].NumSaldaturaAtt;
      L     0;
      ==I;
      );
      JNB   _136;
      L     "DBWork".CoordSaldatura[1].X2;
      T     "MD588";
      SET;
      SAVE;
      CLR;
_136: A     BR;
      );
      JNB   _137;
      L     "DBWork".CoordSaldatura[1].Y2;
      T     "MD592";
_137: NOP   0;
      A(;
      A     L 1.0;
      A(;
      L     "DBWork".PP[1].NumSaldaturaAtt;
      L     1;
      ==I;
      );
      JNB   _138;
      L     "DBWork".CoordSaldatura[2].X2;
      T     "MD588";
      SET;
      SAVE;
      CLR;
_138: A     BR;
      );
      JNB   _139;
      L     "DBWork".CoordSaldatura[2].Y2;
      T     "MD592";
_139: NOP   0;
      A(;
      A     L 1.0;
      A(;
      L     "DBWork".PP[1].NumSaldaturaAtt;
      L     2;
      ==I;
      );
      JNB   _13a;
      L     "DBWork".CoordSaldatura[3].X2;
      T     "MD588";
      SET;
      SAVE;
      CLR;
_13a: A     BR;
      );
      JNB   _13b;
      L     "DBWork".CoordSaldatura[3].Y2;
      T     "MD592";
_13b: NOP   0;
      A(;
      A     L 1.0;
      A(;
      L     "DBWork".PP[1].NumSaldaturaAtt;
      L     3;
      ==I;
      );
      JNB   _13c;
      L     "DBWork".CoordSaldatura[4].X2;
      T     "MD588";
      SET;
      SAVE;
      CLR;
_13c: A     BR;
      );
      JNB   _13d;
      L     "DBWork".CoordSaldatura[4].Y2;
      T     "MD592";
_13d: NOP   0;
      A(;
      A     L 1.0;
      A(;
      L     "DBWork".PP[1].NumSaldaturaAtt;
      L     4;
      ==I;
      );
      JNB   _13e;
      L     "DBWork".CoordSaldatura[5].X2;
      T     "MD588";
      SET;
      SAVE;
      CLR;
_13e: A     BR;
      );
      JNB   _13f;
      L     "DBWork".CoordSaldatura[5].Y2;
      T     "MD592";
_13f: NOP   0;
      A(;
      A     L 1.0;
      A(;
      L     "DBWork".PP[1].NumSaldaturaAtt;
      L     5;
      ==I;
      );
      JNB   _140;
      L     "DBWork".CoordSaldatura[6].X2;
      T     "MD588";
      SET;
      SAVE;
      CLR;
_140: A     BR;
      );
      JNB   _141;
      L     "DBWork".CoordSaldatura[6].Y2;
      T     "MD592";
_141: NOP   0;
      A(;
      A     L 1.0;
      A(;
      L     "DBWork".PP[1].NumSaldaturaAtt;
      L     6;
      ==I;
      );
      JNB   _142;
      L     "DBWork".CoordSaldatura[7].X2;
      T     "MD588";
      SET;
      SAVE;
      CLR;
_142: A     BR;
      );
      JNB   _143;
      L     "DBWork".CoordSaldatura[7].Y2;
      T     "MD592";
_143: NOP   0;
      A(;
      A     L 1.0;
      A(;
      L     "DBWork".PP[1].NumSaldaturaAtt;
      L     7;
      ==I;
      );
      JNB   _144;
      L     "DBWork".CoordSaldatura[8].X2;
      T     "MD588";
      SET;
      SAVE;
      CLR;
_144: A     BR;
      );
      JNB   _145;
      L     "DBWork".CoordSaldatura[8].Y2;
      T     "MD592";
_145: NOP   0;
      A(;
      A     L 1.0;
      A(;
      L     "DBWork".PP[1].NumSaldaturaAtt;
      L     8;
      ==I;
      );
      JNB   _146;
      L     "DBWork".CoordSaldatura[9].X2;
      T     "MD588";
      SET;
      SAVE;
      CLR;
_146: A     BR;
      );
      JNB   _147;
      L     "DBWork".CoordSaldatura[9].Y2;
      T     "MD592";
_147: NOP   0;
      A(;
      A     L 1.0;
      A(;
      L     "DBWork".PP[1].NumSaldaturaAtt;
      L     9;
      ==I;
      );
      JNB   _148;
      L     "DBWork".CoordSaldatura[10].X2;
      T     "MD588";
      SET;
      SAVE;
      CLR;
_148: A     BR;
      );
      JNB   _149;
      L     "DBWork".CoordSaldatura[10].Y2;
      T     "MD592";
_149: NOP   0;
      A(;
      A     L 1.0;
      A(;
      L     "DBWork".PP[1].NumSaldaturaAtt;
      L     10;
      ==I;
      );
      JNB   _14a;
      L     "DBWork".CoordSaldatura[11].X2;
      T     "MD588";
      SET;
      SAVE;
      CLR;
_14a: A     BR;
      );
      JNB   _14b;
      L     "DBWork".CoordSaldatura[11].Y2;
      T     "MD592";
_14b: NOP   0;
      A(;
      A     L 1.0;
      A(;
      L     "DBWork".PP[1].NumSaldaturaAtt;
      L     11;
      ==I;
      );
      JNB   _14c;
      L     "DBWork".CoordSaldatura[12].X2;
      T     "MD588";
      SET;
      SAVE;
      CLR;
_14c: A     BR;
      );
      JNB   _14d;
      L     "DBWork".CoordSaldatura[12].Y2;
      T     "MD592";
_14d: NOP   0;
      A(;
      A     L 1.0;
      A(;
      L     "DBWork".PP[1].NumSaldaturaAtt;
      L     12;
      ==I;
      );
      JNB   _14e;
      L     "DBWork".CoordSaldatura[13].X2;
      T     "MD588";
      SET;
      SAVE;
      CLR;
_14e: A     BR;
      );
      JNB   _14f;
      L     "DBWork".CoordSaldatura[13].Y2;
      T     "MD592";
_14f: NOP   0;
NETWORK
TITLE = ******************** Point for Vision **************************
END_FUNCTION

FUNCTION "FC52 - SYSTEM VISION" : VOID	// FC 52
VERSION : 0.1
BEGIN
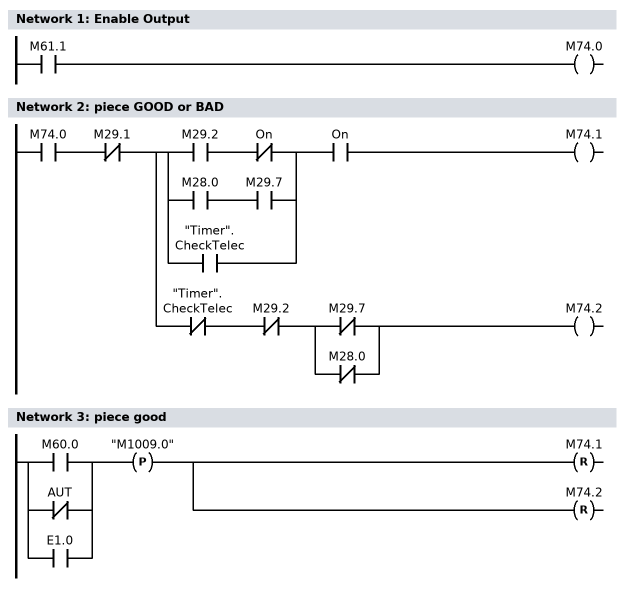
NETWORK
TITLE = Enable Output 
      A     "M61.1";
      =     "M74.0";
NETWORK
TITLE = piece GOOD or BAD
      A     "M74.0";
      AN    "M29.1";
      =     L 0.0;
      A     L 0.0;
      A(;
      A     "M29.2";
      AN    "On";
      O;
      A     "M28.0";
      A     "M29.7";
      O     "Timer".CheckTelec;
      );
      A     "On";
      =     "M74.1";
      A     L 0.0;
      AN    "Timer".CheckTelec;
      AN    "M29.2";
      A(;
      ON    "M29.7";
      ON    "M28.0";
      );
      =     "M74.2";
NETWORK
TITLE = piece good
      A(;
      O     "M60.0";
      ON    "AUT";
      O     "E1.0";
      );
      FP    "M1009.0";
      R     "M74.1";
      R     "M74.2";
END_FUNCTION

